LIN {X 0,Y 216.789,Z 515.517,A -85,B 0,C 180,E1 -25716.63,E2 -25716.63} C_VEL
LIN {X 0,Y 214.368,Z 508.219,A -85,B 0,C 180,E1 -25719.47,E2 -25719.47} C_VEL
LIN {X 0,Y 212.087,Z 502.265,A -85,B 0,C 180,E1 -25722.649,E2 -25722.649} C_VEL
LIN {X 0,Y 210.813,Z 499.684,A -85,B 0,C 180,E1 -25724.747,E2 -25724.747} C_VEL
LIN {X 0,Y 209.329,Z 496.442,A -85,B 0,C 180,E1 -25728.011,E2 -25728.011} C_VEL
LIN {X 0,Y 208.054,Z 493.301,A -85,B 0,C 180,E1 -25734.185,E2 -25734.185} C_VEL
LIN {X 0,Y 208.091,Z 492.674,A -85,B 0,C 180,E1 -25735.157,E2 -25735.157} C_VEL
LIN {X 0,Y 208.128,Z 492.743,A -85,B 0,C 180,E1 -25736.371,E2 -25736.371} C_VEL
LIN {X 0,Y 208.764,Z 495.592,A -85,B 0,C 180,E1 -25740.845,E2 -25740.845} C_VEL
LIN {X 0,Y 209.557,Z 496.767,A -85,B 0,C 180,E1 -25743.005,E2 -25743.005} C_VEL
LIN {X 0,Y 211.535,Z 500.908,A -85,B 0,C 180,E1 -25746.918,E2 -25746.918} C_VEL
LIN {X 0,Y 213.432,Z 504.886,A -85,B 0,C 180,E1 -25749.672,E2 -25749.672} C_VEL
LIN {X 0,Y 216.61,Z 511.711,A -85,B 0,C 180,E1 -25753.307,E2 -25753.307} C_VEL
LIN {X 0,Y 216.993,Z 512.62,A -85,B 0,C 180,E1 -25753.702,E2 -25753.702} C_VEL
LIN {X 0,Y 213.346,Z 546.935,A -85,B 0,C 180,E1 -25754.491,E2 -25754.491} C_VEL
LIN {X 0,Y 210.473,Z 562.769,A -85,B 0,C 180,E1 -25755.095,E2 -25755.095} C_VEL
LIN {X 0,Y 206.526,Z 577.358,A -85,B 0,C 180,E1 -25755.798,E2 -25755.798} C_VEL
LIN {X 0,Y 201.851,Z 590.9,A -85,B 0,C 180,E1 -25756.766,E2 -25756.766} C_VEL
LIN {X 0,Y 195.793,Z 604.759,A -85,B 0,C 180,E1 -25757.969,E2 -25757.969} C_VEL
LIN {X 0,Y 188.994,Z 617.85,A -85,B 0,C 180,E1 -25759.554,E2 -25759.554} C_VEL
LIN {X 0,Y 181.962,Z 629.225,A -85,B 0,C 180,E1 -25761.284,E2 -25761.284} C_VEL
LIN {X 0,Y 174.302,Z 639.946,A -85,B 0,C 180,E1 -25763.358,E2 -25763.358} C_VEL
LIN {X 0,Y 166.007,Z 650.074,A -85,B 0,C 180,E1 -25765.89,E2 -25765.89} C_VEL
LIN {X 0,Y 158.032,Z 658.675,A -85,B 0,C 180,E1 -25768.692,E2 -25768.692} C_VEL
LIN {X 0,Y 149.549,Z 666.826,A -85,B 0,C 180,E1 -25772.231,E2 -25772.231} C_VEL
LIN {X 0,Y 140.342,Z 674.616,A -85,B 0,C 180,E1 -25776.938,E2 -25776.938} C_VEL
LIN {X 0,Y 132.458,Z 680.534,A -85,B 0,C 180,E1 -25782.028,E2 -25782.028} C_VEL
LIN {X 0,Y 125.577,Z 685.126,A -85,B 0,C 180,E1 -25787.81,E2 -25787.81} C_VEL
LIN {X 0,Y 120.021,Z 688.366,A -85,B 0,C 180,E1 -25794.157,E2 -25794.157} C_VEL
LIN {X 0,Y 115.906,Z 690.342,A -85,B 0,C 180,E1 -25800.982,E2 -25800.982} C_VEL
LIN {X 0,Y 113.241,Z 691.138,A -85,B 0,C 180,E1 -25808.586,E2 -25808.586} C_VEL
LIN {X 0,Y 112.042,Z 690.745,A -85,B 0,C 180,E1 -25815.469,E2 -25815.469} C_VEL
LIN {X 0,Y 111.999,Z 689.219,A -85,B 0,C 180,E1 -25822.791,E2 -25822.791} C_VEL
LIN {X 0,Y 112.58,Z 687.675,A -85,B 0,C 180,E1 -25827.259,E2 -25827.259} C_VEL
LIN {X 0,Y 113.611,Z 684.748,A -85,B 0,C 180,E1 -25833.547,E2 -25833.547} C_VEL
LIN {X 0,Y 115.984,Z 680.196,A -85,B 0,C 180,E1 -25840.474,E2 -25840.474} C_VEL
LIN {X 0,Y 119.742,Z 674.292,A -85,B 0,C 180,E1 -25847.066,E2 -25847.066} C_VEL
LIN {X 0,Y 124.77,Z 666.872,A -85,B 0,C 180,E1 -25853.222,E2 -25853.222} C_VEL
LIN {X 0,Y 130.986,Z 657.702,A -85,B 0,C 180,E1 -25858.875,E2 -25858.875} C_VEL
LIN {X 0,Y 137.317,Z 647.92,A -85,B 0,C 180,E1 -25863.381,E2 -25863.381} C_VEL
LIN {X 0,Y 143.335,Z 637.901,A -85,B 0,C 180,E1 -25866.916,E2 -25866.916} C_VEL
LIN {X 0,Y 149.792,Z 626.003,A -85,B 0,C 180,E1 -25870.175,E2 -25870.175} C_VEL
LIN {X 0,Y 155.513,Z 614.116,A -85,B 0,C 180,E1 -25872.679,E2 -25872.679} C_VEL
LIN {X 0,Y 160.824,Z 601.272,A -85,B 0,C 180,E1 -25874.803,E2 -25874.803} C_VEL
LIN {X 0,Y 165.697,Z 587.197,A -85,B 0,C 180,E1 -25876.582,E2 -25876.582} C_VEL
LIN {X 0,Y 169.701,Z 572.604,A -85,B 0,C 180,E1 -25877.976,E2 -25877.976} C_VEL
LIN {X 0,Y 172.855,Z 557.467,A -85,B 0,C 180,E1 -25879.001,E2 -25879.001} C_VEL
LIN {X 0,Y 174.998,Z 541.593,A -85,B 0,C 180,E1 -25879.734,E2 -25879.734} C_VEL
LIN {X 0,Y 180.049,Z 484.1,A -85,B 0,C 180,E1 -25881.46,E2 -25881.46} C_VEL
LIN {X 0,Y 175.965,Z 475.406,A -85,B 0,C 180,E1 -25884.258,E2 -25884.258} C_VEL
LIN {X 0,Y 171.404,Z 466.555,A -85,B 0,C 180,E1 -25887.788,E2 -25887.788} C_VEL
LIN {X 0,Y 167.025,Z 458.934,A -85,B 0,C 180,E1 -25891.77,E2 -25891.77} C_VEL
LIN {X 0,Y 164.311,Z 454.695,A -85,B 0,C 180,E1 -25894.675,E2 -25894.675} C_VEL
LIN {X 0,Y 162.168,Z 451.296,A -85,B 0,C 180,E1 -25897.378,E2 -25897.378} C_VEL
LIN {X 0,Y 159.832,Z 447.476,A -85,B 0,C 180,E1 -25901.022,E2 -25901.022} C_VEL
LIN {X 0,Y 157.239,Z 443.804,A -85,B 0,C 180,E1 -25906.822,E2 -25906.822} C_VEL
LIN {X 0,Y 156.873,Z 442.502,A -85,B 0,C 180,E1 -25908.368,E2 -25908.368} C_VEL
LIN {X 0,Y 155.969,Z 441.952,A -85,B 0,C 180,E1 -25914.828,E2 -25914.828} C_VEL
LIN {X 0,Y 156.825,Z 442.233,A -85,B 0,C 180,E1 -25920.962,E2 -25920.962} C_VEL
LIN {X 0,Y 157.17,Z 442.777,A -85,B 0,C 180,E1 -25922.241,E2 -25922.241} C_VEL
LIN {X 0,Y 158.75,Z 446.055,A -85,B 0,C 180,E1 -25926.553,E2 -25926.553} C_VEL
LIN {X 0,Y 159.904,Z 447.505,A -85,B 0,C 180,E1 -25928.689,E2 -25928.689} C_VEL
LIN {X 0,Y 162.896,Z 452.334,A -85,B 0,C 180,E1 -25933.17,E2 -25933.17} C_VEL
LIN {X 0,Y 165.563,Z 456.628,A -85,B 0,C 180,E1 -25936.318,E2 -25936.318} C_VEL
LIN {X 0,Y 168.544,Z 461.52,A -85,B 0,C 180,E1 -25939.295,E2 -25939.295} C_VEL
LIN {X 0,Y 172.847,Z 469.132,A -85,B 0,C 180,E1 -25942.969,E2 -25942.969} C_VEL
LIN {X 0,Y 174.775,Z 473.432,A -85,B 0,C 180,E1 -25944.498,E2 -25944.498} C_VEL
LIN {X 0,Y 178.254,Z 483.137,A -85,B 0,C 180,E1 -25947.16,E2 -25947.16} C_VEL
LIN {X 0,Y 179.8,Z 487.933,A -85,B 0,C 180,E1 -25948.289,E2 -25948.289} C_VEL
LIN {X 0,Y 174.44,Z 549.298,A -85,B 0,C 180,E1 -25950.164,E2 -25950.164} C_VEL
LIN {X 0,Y 172.197,Z 564.852,A -85,B 0,C 180,E1 -25950.892,E2 -25950.892} C_VEL
LIN {X 0,Y 169.048,Z 579.136,A -85,B 0,C 180,E1 -25951.824,E2 -25951.824} C_VEL
LIN {X 0,Y 164.671,Z 593.902,A -85,B 0,C 180,E1 -25953.114,E2 -25953.114} C_VEL
LIN {X 0,Y 159.805,Z 607.528,A -85,B 0,C 180,E1 -25954.787,E2 -25954.787} C_VEL
LIN {X 0,Y 154.599,Z 619.845,A -85,B 0,C 180,E1 -25956.752,E2 -25956.752} C_VEL
LIN {X 0,Y 148.677,Z 632.077,A -85,B 0,C 180,E1 -25959.281,E2 -25959.281} C_VEL
LIN {X 0,Y 142.549,Z 643.378,A -85,B 0,C 180,E1 -25962.308,E2 -25962.308} C_VEL
LIN {X 0,Y 136.125,Z 654.072,A -85,B 0,C 180,E1 -25966.019,E2 -25966.019} C_VEL
LIN {X 0,Y 129.927,Z 663.892,A -85,B 0,C 180,E1 -25970.536,E2 -25970.536} C_VEL
LIN {X 0,Y 124.282,Z 672.283,A -85,B 0,C 180,E1 -25975.563,E2 -25975.563} C_VEL
LIN {X 0,Y 119.118,Z 680.145,A -85,B 0,C 180,E1 -25981.835,E2 -25981.835} C_VEL
LIN {X 0,Y 115.38,Z 686.373,A -85,B 0,C 180,E1 -25988.563,E2 -25988.563} C_VEL
LIN {X 0,Y 113.13,Z 691.156,A -85,B 0,C 180,E1 -25995.611,E2 -25995.611} C_VEL
LIN {X 0,Y 112.299,Z 693.751,A -85,B 0,C 180,E1 -26000.822,E2 -26000.822} C_VEL
LIN {X 0,Y 111.839,Z 694.596,A -85,B 0,C 180,E1 -26002.781,E2 -26002.781} C_VEL
LIN {X 0,Y 110.357,Z 695.619,A -85,B 0,C 180,E1 -26005.7,E2 -26005.7} C_VEL
LIN {X 0,Y 106.025,Z 697.111,A -85,B 0,C 180,E1 -26012.749,E2 -26012.749} C_VEL
LIN {X 0,Y 105.075,Z 697.517,A -85,B 0,C 180,E1 -26017.077,E2 -26017.077} C_VEL
LIN {X 0,Y 106.25,Z 697.472,A -85,B 0,C 180,E1 -26025.342,E2 -26025.342} C_VEL
LIN {X 0,Y 109.033,Z 696.206,A -85,B 0,C 180,E1 -26032.752,E2 -26032.752} C_VEL
LIN {X 0,Y 113.321,Z 693.824,A -85,B 0,C 180,E1 -26039.745,E2 -26039.745} C_VEL
LIN {X 0,Y 119.308,Z 690.289,A -85,B 0,C 180,E1 -26046.091,E2 -26046.091} C_VEL
LIN {X 0,Y 126.508,Z 685.508,A -85,B 0,C 180,E1 -26051.809,E2 -26051.809} C_VEL
LIN {X 0,Y 134.882,Z 679.357,A -85,B 0,C 180,E1 -26056.842,E2 -26056.842} C_VEL
LIN {X 0,Y 144.149,Z 671.666,A -85,B 0,C 180,E1 -26061.268,E2 -26061.268} C_VEL
LIN {X 0,Y 153.008,Z 663.486,A -85,B 0,C 180,E1 -26064.617,E2 -26064.617} C_VEL
LIN {X 0,Y 162.322,Z 653.69,A -85,B 0,C 180,E1 -26067.596,E2 -26067.596} C_VEL
LIN {X 0,Y 170.695,Z 643.685,A -85,B 0,C 180,E1 -26069.84,E2 -26069.84} C_VEL
LIN {X 0,Y 179.17,Z 631.906,A -85,B 0,C 180,E1 -26071.921,E2 -26071.921} C_VEL
LIN {X 0,Y 186.548,Z 620.052,A -85,B 0,C 180,E1 -26073.478,E2 -26073.478} C_VEL
LIN {X 0,Y 193.259,Z 607.331,A -85,B 0,C 180,E1 -26074.769,E2 -26074.769} C_VEL
LIN {X 0,Y 199.356,Z 593.456,A -85,B 0,C 180,E1 -26075.809,E2 -26075.809} C_VEL
LIN {X 0,Y 204.396,Z 579.169,A -85,B 0,C 180,E1 -26076.582,E2 -26076.582} C_VEL
LIN {X 0,Y 208.074,Z 565.488,A -85,B 0,C 180,E1 -26077.146,E2 -26077.146} C_VEL
LIN {X 0,Y 210.918,Z 549.998,A -85,B 0,C 180,E1 -26077.622,E2 -26077.622} C_VEL
LIN {X 0,Y 214.201,Z 519.191,A -85,B 0,C 180,E1 -26078.355,E2 -26078.355} C_VEL
LIN {X 0,Y 212.313,Z 513.341,A -85,B 0,C 180,E1 -26080.838,E2 -26080.838} C_VEL
LIN {X 0,Y 210.682,Z 508.732,A -85,B 0,C 180,E1 -26083.373,E2 -26083.373} C_VEL
LIN {X 0,Y 209.529,Z 506.271,A -85,B 0,C 180,E1 -26085.431,E2 -26085.431} C_VEL
LIN {X 0,Y 208.189,Z 503.256,A -85,B 0,C 180,E1 -26088.665,E2 -26088.665} C_VEL
LIN {X 0,Y 207.191,Z 500.002,A -85,B 0,C 180,E1 -26094.891,E2 -26094.891} C_VEL
LIN {X 0,Y 207.241,Z 499.914,A -85,B 0,C 180,E1 -26096.355,E2 -26096.355} C_VEL
LIN {X 0,Y 207.883,Z 502.7,A -85,B 0,C 180,E1 -26100.848,E2 -26100.848} C_VEL
LIN {X 0,Y 208.552,Z 503.807,A -85,B 0,C 180,E1 -26102.747,E2 -26102.747} C_VEL
LIN {X 0,Y 210.268,Z 507.604,A -85,B 0,C 180,E1 -26106.358,E2 -26106.358} C_VEL
LIN {X 0,Y 211.925,Z 511.286,A -85,B 0,C 180,E1 -26108.944,E2 -26108.944} C_VEL
LIN {X 0,Y 214.366,Z 516.868,A -85,B 0,C 180,E1 -26111.995,E2 -26111.995} C_VEL
LIN {X 0,Y 210.93,Z 547.937,A -85,B 0,C 180,E1 -26112.704,E2 -26112.704} C_VEL
LIN {X 0,Y 208.048,Z 563.218,A -85,B 0,C 180,E1 -26113.27,E2 -26113.27} C_VEL
LIN {X 0,Y 203.997,Z 577.848,A -85,B 0,C 180,E1 -26113.956,E2 -26113.956} C_VEL
LIN {X 0,Y 199.094,Z 591.641,A -85,B 0,C 180,E1 -26114.909,E2 -26114.909} C_VEL
LIN {X 0,Y 192.901,Z 605.395,A -85,B 0,C 180,E1 -26116.07,E2 -26116.07} C_VEL
LIN {X 0,Y 185.946,Z 618.371,A -85,B 0,C 180,E1 -26117.601,E2 -26117.601} C_VEL
LIN {X 0,Y 178.695,Z 629.723,A -85,B 0,C 180,E1 -26119.281,E2 -26119.281} C_VEL
LIN {X 0,Y 170.492,Z 640.806,A -85,B 0,C 180,E1 -26121.393,E2 -26121.393} C_VEL
LIN {X 0,Y 161.547,Z 651.244,A -85,B 0,C 180,E1 -26123.993,E2 -26123.993} C_VEL
LIN {X 0,Y 152.151,Z 660.809,A -85,B 0,C 180,E1 -26127.23,E2 -26127.23} C_VEL
LIN {X 0,Y 143.274,Z 668.711,A -85,B 0,C 180,E1 -26130.86,E2 -26130.86} C_VEL
LIN {X 0,Y 135.286,Z 675.069,A -85,B 0,C 180,E1 -26134.853,E2 -26134.853} C_VEL
LIN {X 0,Y 127.621,Z 680.518,A -85,B 0,C 180,E1 -26139.559,E2 -26139.559} C_VEL
LIN {X 0,Y 120.208,Z 685.162,A -85,B 0,C 180,E1 -26145.446,E2 -26145.446} C_VEL
LIN {X 0,Y 114.115,Z 688.45,A -85,B 0,C 180,E1 -26151.985,E2 -26151.985} C_VEL
LIN {X 0,Y 109.539,Z 690.489,A -85,B 0,C 180,E1 -26159.118,E2 -26159.118} C_VEL
LIN {X 0,Y 106.295,Z 691.369,A -85,B 0,C 180,E1 -26167.772,E2 -26167.772} C_VEL
LIN {X 0,Y 105.042,Z 691.015,A -85,B 0,C 180,E1 -26174.477,E2 -26174.477} C_VEL
LIN {X 0,Y 104.859,Z 689.549,A -85,B 0,C 180,E1 -26182.297,E2 -26182.297} C_VEL
LIN {X 0,Y 105.519,Z 687.844,A -85,B 0,C 180,E1 -26187.568,E2 -26187.568} C_VEL
LIN {X 0,Y 107.003,Z 684.119,A -85,B 0,C 180,E1 -26195.654,E2 -26195.654} C_VEL
LIN {X 0,Y 109.917,Z 679.324,A -85,B 0,C 180,E1 -26202.932,E2 -26202.932} C_VEL
LIN {X 0,Y 114.167,Z 673.145,A -85,B 0,C 180,E1 -26209.79,E2 -26209.79} C_VEL
LIN {X 0,Y 119.837,Z 665.382,A -85,B 0,C 180,E1 -26216.094,E2 -26216.094} C_VEL
LIN {X 0,Y 125.75,Z 657.124,A -85,B 0,C 180,E1 -26221.13,E2 -26221.13} C_VEL
LIN {X 0,Y 132.488,Z 647.183,A -85,B 0,C 180,E1 -26225.698,E2 -26225.698} C_VEL
LIN {X 0,Y 138.858,Z 637.022,A -85,B 0,C 180,E1 -26229.247,E2 -26229.247} C_VEL
LIN {X 0,Y 145.635,Z 624.903,A -85,B 0,C 180,E1 -26232.502,E2 -26232.502} C_VEL
LIN {X 0,Y 152.228,Z 611.414,A -85,B 0,C 180,E1 -26235.221,E2 -26235.221} C_VEL
LIN {X 0,Y 157.794,Z 597.924,A -85,B 0,C 180,E1 -26237.299,E2 -26237.299} C_VEL
LIN {X 0,Y 162.516,Z 583.963,A -85,B 0,C 180,E1 -26238.946,E2 -26238.946} C_VEL
LIN {X 0,Y 166.4,Z 569.598,A -85,B 0,C 180,E1 -26240.189,E2 -26240.189} C_VEL
LIN {X 0,Y 169.465,Z 554.058,A -85,B 0,C 180,E1 -26241.159,E2 -26241.159} C_VEL
LIN {X 0,Y 171.416,Z 538.62,A -85,B 0,C 180,E1 -26241.773,E2 -26241.773} C_VEL
LIN {X 0,Y 175.994,Z 487.072,A -85,B 0,C 180,E1 -26243.323,E2 -26243.323} C_VEL
LIN {X 0,Y 172.455,Z 479.342,A -85,B 0,C 180,E1 -26245.982,E2 -26245.982} C_VEL
LIN {X 0,Y 168.495,Z 471.452,A -85,B 0,C 180,E1 -26249.338,E2 -26249.338} C_VEL
LIN {X 0,Y 164.672,Z 464.588,A -85,B 0,C 180,E1 -26253.133,E2 -26253.133} C_VEL
LIN {X 0,Y 162.514,Z 461.004,A -85,B 0,C 180,E1 -26255.64,E2 -26255.64} C_VEL
LIN {X 0,Y 160.524,Z 457.695,A -85,B 0,C 180,E1 -26258.347,E2 -26258.347} C_VEL
LIN {X 0,Y 158.412,Z 454.115,A -85,B 0,C 180,E1 -26261.906,E2 -26261.906} C_VEL
LIN {X 0,Y 156.152,Z 450.578,A -85,B 0,C 180,E1 -26267.489,E2 -26267.489} C_VEL
LIN {X 0,Y 155.842,Z 449.447,A -85,B 0,C 180,E1 -26268.949,E2 -26268.949} C_VEL
LIN {X 0,Y 155.264,Z 448.928,A -85,B 0,C 180,E1 -26277.404,E2 -26277.404} C_VEL
LIN {X 0,Y 156.04,Z 449.33,A -85,B 0,C 180,E1 -26281.289,E2 -26281.289} C_VEL
LIN {X 0,Y 157.476,Z 452.718,A -85,B 0,C 180,E1 -26285.762,E2 -26285.762} C_VEL
LIN {X 0,Y 158.654,Z 454.353,A -85,B 0,C 180,E1 -26288.116,E2 -26288.116} C_VEL
LIN {X 0,Y 161.389,Z 459.036,A -85,B 0,C 180,E1 -26292.469,E2 -26292.469} C_VEL
LIN {X 0,Y 163.92,Z 463.28,A -85,B 0,C 180,E1 -26295.622,E2 -26295.622} C_VEL
LIN {X 0,Y 167.147,Z 468.9,A -85,B 0,C 180,E1 -26298.99,E2 -26298.99} C_VEL
LIN {X 0,Y 171,Z 476.238,A -85,B 0,C 180,E1 -26302.423,E2 -26302.423} C_VEL
LIN {X 0,Y 174.282,Z 485.477,A -85,B 0,C 180,E1 -26305.199,E2 -26305.199} C_VEL
LIN {X 0,Y 175.775,Z 490.371,A -85,B 0,C 180,E1 -26306.41,E2 -26306.41} C_VEL
LIN {X 0,Y 171.342,Z 540.726,A -85,B 0,C 180,E1 -26307.941,E2 -26307.941} C_VEL
LIN {X 0,Y 169.414,Z 557.45,A -85,B 0,C 180,E1 -26308.561,E2 -26308.561} C_VEL
LIN {X 0,Y 166.412,Z 572.985,A -85,B 0,C 180,E1 -26309.419,E2 -26309.419} C_VEL
LIN {X 0,Y 162.582,Z 587.033,A -85,B 0,C 180,E1 -26310.475,E2 -26310.475} C_VEL
LIN {X 0,Y 158.178,Z 600.069,A -85,B 0,C 180,E1 -26311.816,E2 -26311.816} C_VEL
LIN {X 0,Y 152.961,Z 613.236,A -85,B 0,C 180,E1 -26313.662,E2 -26313.662} C_VEL
LIN {X 0,Y 147.305,Z 625.255,A -85,B 0,C 180,E1 -26315.798,E2 -26315.798} C_VEL
LIN {X 0,Y 140.693,Z 637.61,A -85,B 0,C 180,E1 -26318.692,E2 -26318.692} C_VEL
LIN {X 0,Y 134.437,Z 648.011,A -85,B 0,C 180,E1 -26321.845,E2 -26321.845} C_VEL
LIN {X 0,Y 128.173,Z 657.582,A -85,B 0,C 180,E1 -26325.63,E2 -26325.63} C_VEL
LIN {X 0,Y 121.791,Z 667.045,A -85,B 0,C 180,E1 -26330.597,E2 -26330.597} C_VEL
LIN {X 0,Y 116.134,Z 674.858,A -85,B 0,C 180,E1 -26335.959,E2 -26335.959} C_VEL
LIN {X 0,Y 111.718,Z 681.228,A -85,B 0,C 180,E1 -26341.726,E2 -26341.726} C_VEL
LIN {X 0,Y 107.962,Z 687.25,A -85,B 0,C 180,E1 -26349.02,E2 -26349.02} C_VEL
LIN {X 0,Y 106.204,Z 690.764,A -85,B 0,C 180,E1 -26354.651,E2 -26354.651} C_VEL
LIN {X 0,Y 105.126,Z 694.276,A -85,B 0,C 180,E1 -26362.316,E2 -26362.316} C_VEL
LIN {X 0,Y 105.08,Z 695.56,A -85,B 0,C 180,E1 -26366.165,E2 -26366.165} C_VEL
LIN {X 0,Y 105.229,Z 696.538,A -85,B 0,C 180,E1 -26370,E2 -26370} C_VEL
LIN {X 0,Y 105.075,Z 697.517,A -85,B 0,C 180,E1 -26377.077,E2 -26377.077} C_VEL
LIN {X 0,Y 104.69,Z 697.712,A -85,B 0,C 180,E1 -26380.291,E2 -26380.291} C_VEL
LIN {X 0,Y 102.814,Z 697.532,A -85,B 0,C 180,E1 -26385.668,E2 -26385.668} C_VEL
LIN {X 0,Y 101.74,Z 696.955,A -85,B 0,C 180,E1 -26390.087,E2 -26390.087} C_VEL
LIN {X 0,Y 102.088,Z 696.277,A -85,B 0,C 180,E1 -26393.399,E2 -26393.399} C_VEL
LIN {X 0,Y 102.536,Z 696.006,A -85,B 0,C 180,E1 -26394.468,E2 -26394.468} C_VEL
LIN {X 0,Y 107.178,Z 693.724,A -85,B 0,C 180,E1 -26401.64,E2 -26401.64} C_VEL
LIN {X 0,Y 113.605,Z 690.245,A -85,B 0,C 180,E1 -26408.216,E2 -26408.216} C_VEL
LIN {X 0,Y 121.286,Z 685.524,A -85,B 0,C 180,E1 -26414.055,E2 -26414.055} C_VEL
LIN {X 0,Y 130.098,Z 679.424,A -85,B 0,C 180,E1 -26419.138,E2 -26419.138} C_VEL
LIN {X 0,Y 139.809,Z 671.801,A -85,B 0,C 180,E1 -26423.542,E2 -26423.542} C_VEL
LIN {X 0,Y 149,Z 663.673,A -85,B 0,C 180,E1 -26426.848,E2 -26426.848} C_VEL
LIN {X 0,Y 158.638,Z 653.96,A -85,B 0,C 180,E1 -26429.756,E2 -26429.756} C_VEL
LIN {X 0,Y 167.252,Z 644.052,A -85,B 0,C 180,E1 -26431.937,E2 -26431.937} C_VEL
LIN {X 0,Y 176.207,Z 632.006,A -85,B 0,C 180,E1 -26434.021,E2 -26434.021} C_VEL
LIN {X 0,Y 184.274,Z 619.396,A -85,B 0,C 180,E1 -26435.584,E2 -26435.584} C_VEL
LIN {X 0,Y 191.125,Z 606.582,A -85,B 0,C 180,E1 -26436.823,E2 -26436.823} C_VEL
LIN {X 0,Y 197.359,Z 592.568,A -85,B 0,C 180,E1 -26437.799,E2 -26437.799} C_VEL
LIN {X 0,Y 202.489,Z 578.078,A -85,B 0,C 180,E1 -26438.53,E2 -26438.53} C_VEL
LIN {X 0,Y 206.431,Z 563.112,A -85,B 0,C 180,E1 -26439.098,E2 -26439.098} C_VEL
LIN {X 0,Y 209.203,Z 547.133,A -85,B 0,C 180,E1 -26439.546,E2 -26439.546} C_VEL
LIN {X 0,Y 211.818,Z 523.026,A -85,B 0,C 180,E1 -26440.093,E2 -26440.093} C_VEL
LIN {X 0,Y 210.195,Z 517.831,A -85,B 0,C 180,E1 -26442.551,E2 -26442.551} C_VEL
LIN {X 0,Y 209.151,Z 514.767,A -85,B 0,C 180,E1 -26444.407,E2 -26444.407} C_VEL
LIN {X 0,Y 208.02,Z 512.33,A -85,B 0,C 180,E1 -26446.694,E2 -26446.694} C_VEL
LIN {X 0,Y 207.182,Z 510.194,A -85,B 0,C 180,E1 -26449.017,E2 -26449.017} C_VEL
LIN {X 0,Y 206.32,Z 507.013,A -85,B 0,C 180,E1 -26455.116,E2 -26455.116} C_VEL
LIN {X 0,Y 206.351,Z 507.112,A -85,B 0,C 180,E1 -26456.339,E2 -26456.339} C_VEL
LIN {X 0,Y 207.117,Z 509.982,A -85,B 0,C 180,E1 -26461.216,E2 -26461.216} C_VEL
LIN {X 0,Y 207.59,Z 510.994,A -85,B 0,C 180,E1 -26462.608,E2 -26462.608} C_VEL
LIN {X 0,Y 209.025,Z 514.28,A -85,B 0,C 180,E1 -26465.79,E2 -26465.79} C_VEL
LIN {X 0,Y 210.584,Z 517.995,A -85,B 0,C 180,E1 -26468.397,E2 -26468.397} C_VEL
LIN {X 0,Y 211.931,Z 521.305,A -85,B 0,C 180,E1 -26470.269,E2 -26470.269} C_VEL
LIN {X 0,Y 208.804,Z 548.452,A -85,B 0,C 180,E1 -26470.867,E2 -26470.867} C_VEL
LIN {X 0,Y 205.723,Z 564.159,A -85,B 0,C 180,E1 -26471.435,E2 -26471.435} C_VEL
LIN {X 0,Y 201.706,Z 578.27,A -85,B 0,C 180,E1 -26472.068,E2 -26472.068} C_VEL
LIN {X 0,Y 196.522,Z 592.439,A -85,B 0,C 180,E1 -26473.009,E2 -26473.009} C_VEL
LIN {X 0,Y 190.228,Z 606.026,A -85,B 0,C 180,E1 -26474.114,E2 -26474.114} C_VEL
LIN {X 0,Y 183.143,Z 618.857,A -85,B 0,C 180,E1 -26475.583,E2 -26475.583} C_VEL
LIN {X 0,Y 174.908,Z 631.315,A -85,B 0,C 180,E1 -26477.388,E2 -26477.388} C_VEL
LIN {X 0,Y 165.97,Z 642.803,A -85,B 0,C 180,E1 -26479.58,E2 -26479.58} C_VEL
LIN {X 0,Y 155.859,Z 653.895,A -85,B 0,C 180,E1 -26482.424,E2 -26482.424} C_VEL
LIN {X 0,Y 146.565,Z 662.751,A -85,B 0,C 180,E1 -26485.568,E2 -26485.568} C_VEL
LIN {X 0,Y 137.116,Z 670.597,A -85,B 0,C 180,E1 -26489.384,E2 -26489.384} C_VEL
LIN {X 0,Y 127.512,Z 677.588,A -85,B 0,C 180,E1 -26494.234,E2 -26494.234} C_VEL
LIN {X 0,Y 118.895,Z 683.012,A -85,B 0,C 180,E1 -26499.786,E2 -26499.786} C_VEL
LIN {X 0,Y 111.529,Z 687.023,A -85,B 0,C 180,E1 -26506.119,E2 -26506.119} C_VEL
LIN {X 0,Y 105.669,Z 689.739,A -85,B 0,C 180,E1 -26513.231,E2 -26513.231} C_VEL
LIN {X 0,Y 101.355,Z 691.238,A -85,B 0,C 180,E1 -26520.963,E2 -26520.963} C_VEL
LIN {X 0,Y 98.808,Z 691.557,A -85,B 0,C 180,E1 -26529.168,E2 -26529.168} C_VEL
LIN {X 0,Y 97.704,Z 690.726,A -85,B 0,C 180,E1 -26537.538,E2 -26537.538} C_VEL
LIN {X 0,Y 98.108,Z 688.727,A -85,B 0,C 180,E1 -26545.892,E2 -26545.892} C_VEL
LIN {X 0,Y 98.662,Z 687.274,A -85,B 0,C 180,E1 -26550,E2 -26550} C_VEL
LIN {X 0,Y 100.537,Z 683.478,A -85,B 0,C 180,E1 -26558.037,E2 -26558.037} C_VEL
LIN {X 0,Y 104.018,Z 678.396,A -85,B 0,C 180,E1 -26565.68,E2 -26565.68} C_VEL
LIN {X 0,Y 108.925,Z 671.906,A -85,B 0,C 180,E1 -26572.776,E2 -26572.776} C_VEL
LIN {X 0,Y 115.202,Z 663.803,A -85,B 0,C 180,E1 -26579.213,E2 -26579.213} C_VEL
LIN {X 0,Y 121.701,Z 655.159,A -85,B 0,C 180,E1 -26584.267,E2 -26584.267} C_VEL
LIN {X 0,Y 128.973,Z 644.774,A -85,B 0,C 180,E1 -26588.805,E2 -26588.805} C_VEL
LIN {X 0,Y 135.763,Z 634.119,A -85,B 0,C 180,E1 -26592.297,E2 -26592.297} C_VEL
LIN {X 0,Y 142.962,Z 621.343,A -85,B 0,C 180,E1 -26595.465,E2 -26595.465} C_VEL
LIN {X 0,Y 149.242,Z 608.44,A -85,B 0,C 180,E1 -26597.876,E2 -26597.876} C_VEL
LIN {X 0,Y 154.401,Z 595.94,A -85,B 0,C 180,E1 -26599.679,E2 -26599.679} C_VEL
LIN {X 0,Y 159.304,Z 581.375,A -85,B 0,C 180,E1 -26601.29,E2 -26601.29} C_VEL
LIN {X 0,Y 163.331,Z 566.08,A -85,B 0,C 180,E1 -26602.5,E2 -26602.5} C_VEL
LIN {X 0,Y 166.173,Z 550.893,A -85,B 0,C 180,E1 -26603.346,E2 -26603.346} C_VEL
LIN {X 0,Y 168.253,Z 532.641,A -85,B 0,C 180,E1 -26603.981,E2 -26603.981} C_VEL
LIN {X 0,Y 172.136,Z 490.174,A -85,B 0,C 180,E1 -26605.253,E2 -26605.253} C_VEL
LIN {X 0,Y 168.053,Z 481.155,A -85,B 0,C 180,E1 -26608.705,E2 -26608.705} C_VEL
LIN {X 0,Y 164.609,Z 474.255,A -85,B 0,C 180,E1 -26612.074,E2 -26612.074} C_VEL
LIN {X 0,Y 161.317,Z 468.144,A -85,B 0,C 180,E1 -26615.917,E2 -26615.917} C_VEL
LIN {X 0,Y 158.955,Z 464.15,A -85,B 0,C 180,E1 -26619.284,E2 -26619.284} C_VEL
LIN {X 0,Y 157.054,Z 460.806,A -85,B 0,C 180,E1 -26622.754,E2 -26622.754} C_VEL
LIN {X 0,Y 155.043,Z 457.148,A -85,B 0,C 180,E1 -26628.395,E2 -26628.395} C_VEL
LIN {X 0,Y 154.824,Z 456.416,A -85,B 0,C 180,E1 -26629.537,E2 -26629.537} C_VEL
LIN {X 0,Y 154.639,Z 456.053,A -85,B 0,C 180,E1 -26639.026,E2 -26639.026} C_VEL
LIN {X 0,Y 155.095,Z 456.555,A -85,B 0,C 180,E1 -26641.135,E2 -26641.135} C_VEL
LIN {X 0,Y 156.731,Z 460.125,A -85,B 0,C 180,E1 -26646.112,E2 -26646.112} C_VEL
LIN {X 0,Y 157.491,Z 461.404,A -85,B 0,C 180,E1 -26647.692,E2 -26647.692} C_VEL
LIN {X 0,Y 159.754,Z 465.419,A -85,B 0,C 180,E1 -26651.525,E2 -26651.525} C_VEL
LIN {X 0,Y 162.225,Z 469.831,A -85,B 0,C 180,E1 -26654.824,E2 -26654.824} C_VEL
LIN {X 0,Y 165.055,Z 475.021,A -85,B 0,C 180,E1 -26657.98,E2 -26657.98} C_VEL
LIN {X 0,Y 168.472,Z 482.034,A -85,B 0,C 180,E1 -26661.267,E2 -26661.267} C_VEL
LIN {X 0,Y 171.375,Z 490.819,A -85,B 0,C 180,E1 -26663.938,E2 -26663.938} C_VEL
LIN {X 0,Y 172.007,Z 493.133,A -85,B 0,C 180,E1 -26664.513,E2 -26664.513} C_VEL
LIN {X 0,Y 166.376,Z 552.178,A -85,B 0,C 180,E1 -26666.284,E2 -26666.284} C_VEL
LIN {X 0,Y 163.719,Z 567.648,A -85,B 0,C 180,E1 -26667.033,E2 -26667.033} C_VEL
LIN {X 0,Y 159.808,Z 583.037,A -85,B 0,C 180,E1 -26668.078,E2 -26668.078} C_VEL
LIN {X 0,Y 155.201,Z 596.864,A -85,B 0,C 180,E1 -26669.343,E2 -26669.343} C_VEL
LIN {X 0,Y 149.688,Z 610.704,A -85,B 0,C 180,E1 -26671.138,E2 -26671.138} C_VEL
LIN {X 0,Y 143.214,Z 624.247,A -85,B 0,C 180,E1 -26673.462,E2 -26673.462} C_VEL
LIN {X 0,Y 136.279,Z 636.732,A -85,B 0,C 180,E1 -26676.313,E2 -26676.313} C_VEL
LIN {X 0,Y 128.599,Z 648.937,A -85,B 0,C 180,E1 -26680.083,E2 -26680.083} C_VEL
LIN {X 0,Y 121.707,Z 658.981,A -85,B 0,C 180,E1 -26684.27,E2 -26684.27} C_VEL
LIN {X 0,Y 115.384,Z 667.676,A -85,B 0,C 180,E1 -26689.097,E2 -26689.097} C_VEL
LIN {X 0,Y 109.48,Z 675.337,A -85,B 0,C 180,E1 -26694.707,E2 -26694.707} C_VEL
LIN {X 0,Y 104.172,Z 682.484,A -85,B 0,C 180,E1 -26701.819,E2 -26701.819} C_VEL
LIN {X 0,Y 100.526,Z 688.094,A -85,B 0,C 180,E1 -26709.539,E2 -26709.539} C_VEL
LIN {X 0,Y 98.483,Z 692.315,A -85,B 0,C 180,E1 -26717.638,E2 -26717.638} C_VEL
LIN {X 0,Y 97.99,Z 695.251,A -85,B 0,C 180,E1 -26725.887,E2 -26725.887} C_VEL
LIN {X 0,Y 98.141,Z 696.256,A -85,B 0,C 180,E1 -26730,E2 -26730} C_VEL
LIN {X 0,Y 97.988,Z 697.242,A -85,B 0,C 180,E1 -26737.192,E2 -26737.192} C_VEL
LIN {X 0,Y 98.507,Z 697.457,A -85,B 0,C 180,E1 -26742.359,E2 -26742.359} C_VEL
LIN {X 0,Y 100.662,Z 696.793,A -85,B 0,C 180,E1 -26750.431,E2 -26750.431} C_VEL
LIN {X 0,Y 102.536,Z 696.006,A -85,B 0,C 180,E1 -26754.468,E2 -26754.468} C_VEL
LIN {X 0,Y 103.673,Z 695.202,A -85,B 0,C 180,E1 -26757.655,E2 -26757.655} C_VEL
LIN {X 0,Y 104.516,Z 693.542,A -85,B 0,C 180,E1 -26763.023,E2 -26763.023} C_VEL
LIN {X 0,Y 105.685,Z 691.951,A -85,B 0,C 180,E1 -26767.217,E2 -26767.217} C_VEL
LIN {X 0,Y 107.622,Z 690.485,A -85,B 0,C 180,E1 -26770.109,E2 -26770.109} C_VEL
LIN {X 0,Y 108.554,Z 689.922,A -85,B 0,C 180,E1 -26770.981,E2 -26770.981} C_VEL
LIN {X 0,Y 116.272,Z 685.529,A -85,B 0,C 180,E1 -26776.497,E2 -26776.497} C_VEL
LIN {X 0,Y 125.539,Z 679.474,A -85,B 0,C 180,E1 -26781.606,E2 -26781.606} C_VEL
LIN {X 0,Y 135.697,Z 671.918,A -85,B 0,C 180,E1 -26785.962,E2 -26785.962} C_VEL
LIN {X 0,Y 146.621,Z 662.624,A -85,B 0,C 180,E1 -26789.632,E2 -26789.632} C_VEL
LIN {X 0,Y 156.632,Z 652.747,A -85,B 0,C 180,E1 -26792.396,E2 -26792.396} C_VEL
LIN {X 0,Y 167.012,Z 640.811,A -85,B 0,C 180,E1 -26794.788,E2 -26794.788} C_VEL
LIN {X 0,Y 176.018,Z 628.482,A -85,B 0,C 180,E1 -26796.684,E2 -26796.684} C_VEL
LIN {X 0,Y 183.818,Z 616.127,A -85,B 0,C 180,E1 -26797.997,E2 -26797.997} C_VEL
LIN {X 0,Y 190.826,Z 602.657,A -85,B 0,C 180,E1 -26799.155,E2 -26799.155} C_VEL
LIN {X 0,Y 196.816,Z 588.708,A -85,B 0,C 180,E1 -26799.981,E2 -26799.981} C_VEL
LIN {X 0,Y 201.952,Z 573.212,A -85,B 0,C 180,E1 -26800.684,E2 -26800.684} C_VEL
LIN {X 0,Y 205.699,Z 557.544,A -85,B 0,C 180,E1 -26801.164,E2 -26801.164} C_VEL
LIN {X 0,Y 208.137,Z 540.924,A -85,B 0,C 180,E1 -26801.546,E2 -26801.546} C_VEL
LIN {X 0,Y 209.602,Z 527.004,A -85,B 0,C 180,E1 -26801.885,E2 -26801.885} C_VEL
LIN {X 0,Y 208.043,Z 521.793,A -85,B 0,C 180,E1 -26804.73,E2 -26804.73} C_VEL
LIN {X 0,Y 207.139,Z 519.636,A -85,B 0,C 180,E1 -26806.637,E2 -26806.637} C_VEL
LIN {X 0,Y 206.242,Z 517.189,A -85,B 0,C 180,E1 -26809.199,E2 -26809.199} C_VEL
LIN {X 0,Y 205.44,Z 514.146,A -85,B 0,C 180,E1 -26815.095,E2 -26815.095} C_VEL
LIN {X 0,Y 205.464,Z 514.361,A -85,B 0,C 180,E1 -26816.446,E2 -26816.446} C_VEL
LIN {X 0,Y 206.237,Z 517.083,A -85,B 0,C 180,E1 -26821.221,E2 -26821.221} C_VEL
LIN {X 0,Y 207.691,Z 520.642,A -85,B 0,C 180,E1 -26824.975,E2 -26824.975} C_VEL
LIN {X 0,Y 209.19,Z 524.506,A -85,B 0,C 180,E1 -26827.724,E2 -26827.724} C_VEL
LIN {X 0,Y 209.662,Z 525.825,A -85,B 0,C 180,E1 -26828.481,E2 -26828.481} C_VEL
LIN {X 0,Y 206.798,Z 549.504,A -85,B 0,C 180,E1 -26829.003,E2 -26829.003} C_VEL
LIN {X 0,Y 203.721,Z 564.642,A -85,B 0,C 180,E1 -26829.527,E2 -26829.527} C_VEL
LIN {X 0,Y 199.579,Z 578.844,A -85,B 0,C 180,E1 -26830.142,E2 -26830.142} C_VEL
LIN {X 0,Y 194.132,Z 593.297,A -85,B 0,C 180,E1 -26831.069,E2 -26831.069} C_VEL
LIN {X 0,Y 187.781,Z 606.64,A -85,B 0,C 180,E1 -26832.104,E2 -26832.104} C_VEL
LIN {X 0,Y 180.522,Z 619.42,A -85,B 0,C 180,E1 -26833.51,E2 -26833.51} C_VEL
LIN {X 0,Y 172.087,Z 631.81,A -85,B 0,C 180,E1 -26835.239,E2 -26835.239} C_VEL
LIN {X 0,Y 163.657,Z 642.346,A -85,B 0,C 180,E1 -26837.158,E2 -26837.158} C_VEL
LIN {X 0,Y 154.686,Z 652.071,A -85,B 0,C 180,E1 -26839.481,E2 -26839.481} C_VEL
LIN {X 0,Y 144.585,Z 661.568,A -85,B 0,C 180,E1 -26842.549,E2 -26842.549} C_VEL
LIN {X 0,Y 134.974,Z 669.413,A -85,B 0,C 180,E1 -26846.078,E2 -26846.078} C_VEL
LIN {X 0,Y 125.805,Z 675.959,A -85,B 0,C 180,E1 -26850.186,E2 -26850.186} C_VEL
LIN {X 0,Y 116.497,Z 681.748,A -85,B 0,C 180,E1 -26855.47,E2 -26855.47} C_VEL
LIN {X 0,Y 110.159,Z 685.207,A -85,B 0,C 180,E1 -26860.041,E2 -26860.041} C_VEL
LIN {X 0,Y 102.876,Z 688.625,A -85,B 0,C 180,E1 -26866.91,E2 -26866.91} C_VEL
LIN {X 0,Y 97.205,Z 690.788,A -85,B 0,C 180,E1 -26874.662,E2 -26874.662} C_VEL
LIN {X 0,Y 93.266,Z 691.754,A -85,B 0,C 180,E1 -26883.12,E2 -26883.12} C_VEL
LIN {X 0,Y 91.138,Z 691.553,A -85,B 0,C 180,E1 -26892.034,E2 -26892.034} C_VEL
LIN {X 0,Y 90.586,Z 690.193,A -85,B 0,C 180,E1 -26901.074,E2 -26901.074} C_VEL
LIN {X 0,Y 91.396,Z 688.104,A -85,B 0,C 180,E1 -26908.562,E2 -26908.562} C_VEL
LIN {X 0,Y 92.918,Z 684.955,A -85,B 0,C 180,E1 -26916.515,E2 -26916.515} C_VEL
LIN {X 0,Y 96.129,Z 680.295,A -85,B 0,C 180,E1 -26924.826,E2 -26924.826} C_VEL
LIN {X 0,Y 100.98,Z 674.247,A -85,B 0,C 180,E1 -26932.507,E2 -26932.507} C_VEL
LIN {X 0,Y 107.306,Z 666.646,A -85,B 0,C 180,E1 -26939.42,E2 -26939.42} C_VEL
LIN {X 0,Y 113.869,Z 658.515,A -85,B 0,C 180,E1 -26944.814,E2 -26944.814} C_VEL
LIN {X 0,Y 121.3,Z 648.761,A -85,B 0,C 180,E1 -26949.593,E2 -26949.593} C_VEL
LIN {X 0,Y 128.251,Z 638.773,A -85,B 0,C 180,E1 -26953.235,E2 -26953.235} C_VEL
LIN {X 0,Y 135.586,Z 626.916,A -85,B 0,C 180,E1 -26956.526,E2 -26956.526} C_VEL
LIN {X 0,Y 142.006,Z 615.08,A -85,B 0,C 180,E1 -26959.003,E2 -26959.003} C_VEL
LIN {X 0,Y 147.948,Z 602.296,A -85,B 0,C 180,E1 -26961.066,E2 -26961.066} C_VEL
LIN {X 0,Y 153.335,Z 588.316,A -85,B 0,C 180,E1 -26962.785,E2 -26962.785} C_VEL
LIN {X 0,Y 157.764,Z 573.859,A -85,B 0,C 180,E1 -26964.117,E2 -26964.117} C_VEL
LIN {X 0,Y 161.388,Z 558.067,A -85,B 0,C 180,E1 -26965.145,E2 -26965.145} C_VEL
LIN {X 0,Y 163.641,Z 543.253,A -85,B 0,C 180,E1 -26965.8,E2 -26965.8} C_VEL
LIN {X 0,Y 168.454,Z 493.301,A -85,B 0,C 180,E1 -26967.285,E2 -26967.285} C_VEL
LIN {X 0,Y 164.508,Z 484.364,A -85,B 0,C 180,E1 -26971.04,E2 -26971.04} C_VEL
LIN {X 0,Y 161.091,Z 477.351,A -85,B 0,C 180,E1 -26974.917,E2 -26974.917} C_VEL
LIN {X 0,Y 158.862,Z 473.239,A -85,B 0,C 180,E1 -26977.935,E2 -26977.935} C_VEL
LIN {X 0,Y 157.601,Z 470.867,A -85,B 0,C 180,E1 -26979.95,E2 -26979.95} C_VEL
LIN {X 0,Y 155.851,Z 467.624,A -85,B 0,C 180,E1 -26983.361,E2 -26983.361} C_VEL
LIN {X 0,Y 153.995,Z 463.881,A -85,B 0,C 180,E1 -26989.148,E2 -26989.148} C_VEL
LIN {X 0,Y 153.811,Z 463.366,A -85,B 0,C 180,E1 -26990.201,E2 -26990.201} C_VEL
LIN {X 0,Y 153.518,Z 463.022,A -85,B 0,C 180,E1 -26997.375,E2 -26997.375} C_VEL
LIN {X 0,Y 154.077,Z 463.423,A -85,B 0,C 180,E1 -27000.551,E2 -27000.551} C_VEL
LIN {X 0,Y 155.698,Z 467.117,A -85,B 0,C 180,E1 -27005.828,E2 -27005.828} C_VEL
LIN {X 0,Y 158.258,Z 471.997,A -85,B 0,C 180,E1 -27010.716,E2 -27010.716} C_VEL
LIN {X 0,Y 160.58,Z 476.391,A -85,B 0,C 180,E1 -27014.029,E2 -27014.029} C_VEL
LIN {X 0,Y 163.378,Z 481.921,A -85,B 0,C 180,E1 -27017.347,E2 -27017.347} C_VEL
LIN {X 0,Y 165.981,Z 487.711,A -85,B 0,C 180,E1 -27020.041,E2 -27020.041} C_VEL
LIN {X 0,Y 168.318,Z 495.35,A -85,B 0,C 180,E1 -27022.407,E2 -27022.407} C_VEL
LIN {X 0,Y 168.171,Z 498.155,A -85,B 0,C 180,E1 -27022.567,E2 -27022.567} C_VEL
LIN {X 0,Y 162.778,Z 552.374,A -85,B 0,C 180,E1 -27024.163,E2 -27024.163} C_VEL
LIN {X 0,Y 160.04,Z 567.707,A -85,B 0,C 180,E1 -27024.892,E2 -27024.892} C_VEL
LIN {X 0,Y 156.212,Z 582.458,A -85,B 0,C 180,E1 -27025.867,E2 -27025.867} C_VEL
LIN {X 0,Y 151.103,Z 597.268,A -85,B 0,C 180,E1 -27027.185,E2 -27027.185} C_VEL
LIN {X 0,Y 145.747,Z 610.227,A -85,B 0,C 180,E1 -27028.828,E2 -27028.828} C_VEL
LIN {X 0,Y 139.357,Z 623.173,A -85,B 0,C 180,E1 -27030.981,E2 -27030.981} C_VEL
LIN {X 0,Y 132.804,Z 634.731,A -85,B 0,C 180,E1 -27033.541,E2 -27033.541} C_VEL
LIN {X 0,Y 125.311,Z 646.388,A -85,B 0,C 180,E1 -27036.945,E2 -27036.945} C_VEL
LIN {X 0,Y 117.923,Z 656.652,A -85,B 0,C 180,E1 -27040.962,E2 -27040.962} C_VEL
LIN {X 0,Y 111.018,Z 665.787,A -85,B 0,C 180,E1 -27045.864,E2 -27045.864} C_VEL
LIN {X 0,Y 104.522,Z 673.752,A -85,B 0,C 180,E1 -27051.54,E2 -27051.54} C_VEL
LIN {X 0,Y 98.589,Z 681.124,A -85,B 0,C 180,E1 -27058.804,E2 -27058.804} C_VEL
LIN {X 0,Y 94.68,Z 686.402,A -85,B 0,C 180,E1 -27065.904,E2 -27065.904} C_VEL
LIN {X 0,Y 92.434,Z 689.974,A -85,B 0,C 180,E1 -27072.294,E2 -27072.294} C_VEL
LIN {X 0,Y 90.995,Z 693.601,A -85,B 0,C 180,E1 -27081.114,E2 -27081.114} C_VEL
LIN {X 0,Y 90.895,Z 694.941,A -85,B 0,C 180,E1 -27085.565,E2 -27085.565} C_VEL
LIN {X 0,Y 91.044,Z 695.973,A -85,B 0,C 180,E1 -27090,E2 -27090} C_VEL
LIN {X 0,Y 91.018,Z 697.109,A -85,B 0,C 180,E1 -27098.884,E2 -27098.884} C_VEL
LIN {X 0,Y 92.522,Z 697.057,A -85,B 0,C 180,E1 -27107.688,E2 -27107.688} C_VEL
LIN {X 0,Y 95.958,Z 695.895,A -85,B 0,C 180,E1 -27116.068,E2 -27116.068} C_VEL
LIN {X 0,Y 101.159,Z 693.623,A -85,B 0,C 180,E1 -27123.766,E2 -27123.766} C_VEL
LIN {X 0,Y 108.554,Z 689.922,A -85,B 0,C 180,E1 -27130.981,E2 -27130.981} C_VEL
LIN {X 0,Y 111.153,Z 688.246,A -85,B 0,C 180,E1 -27133.601,E2 -27133.601} C_VEL
LIN {X 0,Y 114.437,Z 685.213,A -85,B 0,C 180,E1 -27138.108,E2 -27138.108} C_VEL
LIN {X 0,Y 117.327,Z 682.522,A -85,B 0,C 180,E1 -27141.522,E2 -27141.522} C_VEL
LIN {X 0,Y 120.262,Z 680.203,A -85,B 0,C 180,E1 -27143.738,E2 -27143.738} C_VEL
LIN {X 0,Y 121.447,Z 679.363,A -85,B 0,C 180,E1 -27144.372,E2 -27144.372} C_VEL
LIN {X 0,Y 131.838,Z 672.031,A -85,B 0,C 180,E1 -27148.531,E2 -27148.531} C_VEL
LIN {X 0,Y 143.167,Z 662.818,A -85,B 0,C 180,E1 -27152.081,E2 -27152.081} C_VEL
LIN {X 0,Y 153.478,Z 653.021,A -85,B 0,C 180,E1 -27154.74,E2 -27154.74} C_VEL
LIN {X 0,Y 162.598,Z 643.014,A -85,B 0,C 180,E1 -27156.707,E2 -27156.707} C_VEL
LIN {X 0,Y 171.738,Z 631.245,A -85,B 0,C 180,E1 -27158.542,E2 -27158.542} C_VEL
LIN {X 0,Y 179.691,Z 619.372,A -85,B 0,C 180,E1 -27159.831,E2 -27159.831} C_VEL
LIN {X 0,Y 186.831,Z 606.649,A -85,B 0,C 180,E1 -27160.931,E2 -27160.931} C_VEL
LIN {X 0,Y 193.288,Z 592.767,A -85,B 0,C 180,E1 -27161.789,E2 -27161.789} C_VEL
LIN {X 0,Y 198.584,Z 578.484,A -85,B 0,C 180,E1 -27162.428,E2 -27162.428} C_VEL
LIN {X 0,Y 202.534,Z 564.431,A -85,B 0,C 180,E1 -27162.908,E2 -27162.908} C_VEL
LIN {X 0,Y 205.448,Z 549.382,A -85,B 0,C 180,E1 -27163.302,E2 -27163.302} C_VEL
LIN {X 0,Y 207.591,Z 531.323,A -85,B 0,C 180,E1 -27163.682,E2 -27163.682} C_VEL
LIN {X 0,Y 206.633,Z 527.918,A -85,B 0,C 180,E1 -27165.725,E2 -27165.725} C_VEL
LIN {X 0,Y 205.219,Z 524.095,A -85,B 0,C 180,E1 -27169.643,E2 -27169.643} C_VEL
LIN {X 0,Y 204.557,Z 521.295,A -85,B 0,C 180,E1 -27175.11,E2 -27175.11} C_VEL
LIN {X 0,Y 204.577,Z 521.531,A -85,B 0,C 180,E1 -27176.431,E2 -27176.431} C_VEL
LIN {X 0,Y 205.46,Z 524.522,A -85,B 0,C 180,E1 -27181.593,E2 -27181.593} C_VEL
LIN {X 0,Y 206.769,Z 528.107,A -85,B 0,C 180,E1 -27184.998,E2 -27184.998} C_VEL
LIN {X 0,Y 207.624,Z 530.468,A -85,B 0,C 180,E1 -27186.682,E2 -27186.682} C_VEL
LIN {X 0,Y 205.094,Z 550.207,A -85,B 0,C 180,E1 -27187.095,E2 -27187.095} C_VEL
LIN {X 0,Y 201.807,Z 565.756,A -85,B 0,C 180,E1 -27187.625,E2 -27187.625} C_VEL
LIN {X 0,Y 197.722,Z 579.339,A -85,B 0,C 180,E1 -27188.175,E2 -27188.175} C_VEL
LIN {X 0,Y 192.149,Z 593.753,A -85,B 0,C 180,E1 -27189.051,E2 -27189.051} C_VEL
LIN {X 0,Y 185.572,Z 607.238,A -85,B 0,C 180,E1 -27190.043,E2 -27190.043} C_VEL
LIN {X 0,Y 178.171,Z 619.933,A -85,B 0,C 180,E1 -27191.376,E2 -27191.376} C_VEL
LIN {X 0,Y 169.52,Z 632.299,A -85,B 0,C 180,E1 -27193.026,E2 -27193.026} C_VEL
LIN {X 0,Y 160.097,Z 643.695,A -85,B 0,C 180,E1 -27195.036,E2 -27195.036} C_VEL
LIN {X 0,Y 150.875,Z 653.24,A -85,B 0,C 180,E1 -27197.269,E2 -27197.269} C_VEL
LIN {X 0,Y 141.915,Z 661.32,A -85,B 0,C 180,E1 -27199.791,E2 -27199.791} C_VEL
LIN {X 0,Y 131.904,Z 669.253,A -85,B 0,C 180,E1 -27203.205,E2 -27203.205} C_VEL
LIN {X 0,Y 121.423,Z 676.399,A -85,B 0,C 180,E1 -27207.585,E2 -27207.585} C_VEL
LIN {X 0,Y 112.387,Z 681.737,A -85,B 0,C 180,E1 -27212.413,E2 -27212.413} C_VEL
LIN {X 0,Y 105.564,Z 685.23,A -85,B 0,C 180,E1 -27216.974,E2 -27216.974} C_VEL
LIN {X 0,Y 97.614,Z 688.713,A -85,B 0,C 180,E1 -27223.947,E2 -27223.947} C_VEL
LIN {X 0,Y 91.296,Z 690.938,A -85,B 0,C 180,E1 -27231.987,E2 -27231.987} C_VEL
LIN {X 0,Y 86.792,Z 691.965,A -85,B 0,C 180,E1 -27240.932,E2 -27240.932} C_VEL
LIN {X 0,Y 84.256,Z 691.822,A -85,B 0,C 180,E1 -27250.51,E2 -27250.51} C_VEL
LIN {X 0,Y 83.477,Z 690.491,A -85,B 0,C 180,E1 -27260.307,E2 -27260.307} C_VEL
LIN {X 0,Y 84.428,Z 687.983,A -85,B 0,C 180,E1 -27270,E2 -27270} C_VEL
LIN {X 0,Y 86.54,Z 684.308,A -85,B 0,C 180,E1 -27279.348,E2 -27279.348} C_VEL
LIN {X 0,Y 90.438,Z 679.36,A -85,B 0,C 180,E1 -27288.11,E2 -27288.11} C_VEL
LIN {X 0,Y 96.057,Z 673.007,A -85,B 0,C 180,E1 -27296.04,E2 -27296.04} C_VEL
LIN {X 0,Y 103.097,Z 665.062,A -85,B 0,C 180,E1 -27303.049,E2 -27303.049} C_VEL
LIN {X 0,Y 110.305,Z 656.593,A -85,B 0,C 180,E1 -27308.405,E2 -27308.405} C_VEL
LIN {X 0,Y 118.305,Z 646.408,A -85,B 0,C 180,E1 -27313.092,E2 -27313.092} C_VEL
LIN {X 0,Y 125.698,Z 635.989,A -85,B 0,C 180,E1 -27316.624,E2 -27316.624} C_VEL
LIN {X 0,Y 132.799,Z 624.668,A -85,B 0,C 180,E1 -27319.531,E2 -27319.531} C_VEL
LIN {X 0,Y 139.534,Z 612.373,A -85,B 0,C 180,E1 -27321.906,E2 -27321.906} C_VEL
LIN {X 0,Y 145.689,Z 598.959,A -85,B 0,C 180,E1 -27323.903,E2 -27323.903} C_VEL
LIN {X 0,Y 150.929,Z 585.072,A -85,B 0,C 180,E1 -27325.449,E2 -27325.449} C_VEL
LIN {X 0,Y 155.178,Z 570.831,A -85,B 0,C 180,E1 -27326.62,E2 -27326.62} C_VEL
LIN {X 0,Y 158.552,Z 555.519,A -85,B 0,C 180,E1 -27327.525,E2 -27327.525} C_VEL
LIN {X 0,Y 160.658,Z 540.75,A -85,B 0,C 180,E1 -27328.105,E2 -27328.105} C_VEL
LIN {X 0,Y 165.039,Z 496.794,A -85,B 0,C 180,E1 -27329.334,E2 -27329.334} C_VEL
LIN {X 0,Y 161.816,Z 489.085,A -85,B 0,C 180,E1 -27332.778,E2 -27332.778} C_VEL
LIN {X 0,Y 158.845,Z 482.763,A -85,B 0,C 180,E1 -27336.533,E2 -27336.533} C_VEL
LIN {X 0,Y 156.544,Z 478.048,A -85,B 0,C 180,E1 -27340.145,E2 -27340.145} C_VEL
LIN {X 0,Y 154.582,Z 474.351,A -85,B 0,C 180,E1 -27344.169,E2 -27344.169} C_VEL
LIN {X 0,Y 152.946,Z 470.432,A -85,B 0,C 180,E1 -27350.145,E2 -27350.145} C_VEL
LIN {X 0,Y 152.832,Z 470.127,A -85,B 0,C 180,E1 -27358.681,E2 -27358.681} C_VEL
LIN {X 0,Y 153.131,Z 470.584,A -85,B 0,C 180,E1 -27360.334,E2 -27360.334} C_VEL
LIN {X 0,Y 154.941,Z 474.795,A -85,B 0,C 180,E1 -27366.221,E2 -27366.221} C_VEL
LIN {X 0,Y 157.039,Z 479.093,A -85,B 0,C 180,E1 -27370.311,E2 -27370.311} C_VEL
LIN {X 0,Y 159.104,Z 483.21,A -85,B 0,C 180,E1 -27373.408,E2 -27373.408} C_VEL
LIN {X 0,Y 161.939,Z 489.293,A -85,B 0,C 180,E1 -27376.951,E2 -27376.951} C_VEL
LIN {X 0,Y 163.715,Z 493.75,A -85,B 0,C 180,E1 -27378.932,E2 -27378.932} C_VEL
LIN {X 0,Y 164.93,Z 498.179,A -85,B 0,C 180,E1 -27380.32,E2 -27380.32} C_VEL
LIN {X 0,Y 161.379,Z 535.237,A -85,B 0,C 180,E1 -27381.435,E2 -27381.435} C_VEL
LIN {X 0,Y 159.186,Z 553.98,A -85,B 0,C 180,E1 -27382.005,E2 -27382.005} C_VEL
LIN {X 0,Y 156.189,Z 569.282,A -85,B 0,C 180,E1 -27382.715,E2 -27382.715} C_VEL
LIN {X 0,Y 152.087,Z 584.151,A -85,B 0,C 180,E1 -27383.716,E2 -27383.716} C_VEL
LIN {X 0,Y 147.225,Z 597.655,A -85,B 0,C 180,E1 -27384.906,E2 -27384.906} C_VEL
LIN {X 0,Y 141.466,Z 611.039,A -85,B 0,C 180,E1 -27386.589,E2 -27386.589} C_VEL
LIN {X 0,Y 135.098,Z 623.397,A -85,B 0,C 180,E1 -27388.614,E2 -27388.614} C_VEL
LIN {X 0,Y 127.627,Z 635.962,A -85,B 0,C 180,E1 -27391.401,E2 -27391.401} C_VEL
LIN {X 0,Y 119.859,Z 647.382,A -85,B 0,C 180,E1 -27394.824,E2 -27394.824} C_VEL
LIN {X 0,Y 111.798,Z 657.903,A -85,B 0,C 180,E1 -27399.103,E2 -27399.103} C_VEL
LIN {X 0,Y 103.885,Z 667.65,A -85,B 0,C 180,E1 -27404.737,E2 -27404.737} C_VEL
LIN {X 0,Y 96.348,Z 676.227,A -85,B 0,C 180,E1 -27411.682,E2 -27411.682} C_VEL
LIN {X 0,Y 90.449,Z 683.105,A -85,B 0,C 180,E1 -27419.664,E2 -27419.664} C_VEL
LIN {X 0,Y 86.364,Z 688.489,A -85,B 0,C 180,E1 -27428.519,E2 -27428.519} C_VEL
LIN {X 0,Y 84.566,Z 691.58,A -85,B 0,C 180,E1 -27435.562,E2 -27435.562} C_VEL
LIN {X 0,Y 83.792,Z 694.629,A -85,B 0,C 180,E1 -27445.188,E2 -27445.188} C_VEL
LIN {X 0,Y 83.94,Z 695.688,A -85,B 0,C 180,E1 -27450,E2 -27450} C_VEL
LIN {X 0,Y 83.978,Z 696.861,A -85,B 0,C 180,E1 -27459.635,E2 -27459.635} C_VEL
LIN {X 0,Y 85.725,Z 696.849,A -85,B 0,C 180,E1 -27469.143,E2 -27469.143} C_VEL
LIN {X 0,Y 89.568,Z 695.74,A -85,B 0,C 180,E1 -27478.086,E2 -27478.086} C_VEL
LIN {X 0,Y 95.299,Z 693.523,A -85,B 0,C 180,E1 -27486.155,E2 -27486.155} C_VEL
LIN {X 0,Y 102.735,Z 690.156,A -85,B 0,C 180,E1 -27493.164,E2 -27493.164} C_VEL
LIN {X 0,Y 111.486,Z 685.518,A -85,B 0,C 180,E1 -27499.154,E2 -27499.154} C_VEL
LIN {X 0,Y 121.447,Z 679.363,A -85,B 0,C 180,E1 -27504.372,E2 -27504.372} C_VEL
LIN {X 0,Y 124.807,Z 676.811,A -85,B 0,C 180,E1 -27506.3,E2 -27506.3} C_VEL
LIN {X 0,Y 133.396,Z 668.706,A -85,B 0,C 180,E1 -27512.241,E2 -27512.241} C_VEL
LIN {X 0,Y 136.868,Z 665.614,A -85,B 0,C 180,E1 -27513.773,E2 -27513.773} C_VEL
LIN {X 0,Y 138.171,Z 664.491,A -85,B 0,C 180,E1 -27514.18,E2 -27514.18} C_VEL
LIN {X 0,Y 149.052,Z 654.77,A -85,B 0,C 180,E1 -27516.846,E2 -27516.846} C_VEL
LIN {X 0,Y 158.373,Z 645.154,A -85,B 0,C 180,E1 -27518.733,E2 -27518.733} C_VEL
LIN {X 0,Y 168.346,Z 632.986,A -85,B 0,C 180,E1 -27520.616,E2 -27520.616} C_VEL
LIN {X 0,Y 176.576,Z 621.307,A -85,B 0,C 180,E1 -27521.854,E2 -27521.854} C_VEL
LIN {X 0,Y 183.842,Z 609.073,A -85,B 0,C 180,E1 -27522.885,E2 -27522.885} C_VEL
LIN {X 0,Y 190.39,Z 595.817,A -85,B 0,C 180,E1 -27523.69,E2 -27523.69} C_VEL
LIN {X 0,Y 196.176,Z 581.245,A -85,B 0,C 180,E1 -27524.323,E2 -27524.323} C_VEL
LIN {X 0,Y 200.562,Z 566.626,A -85,B 0,C 180,E1 -27524.817,E2 -27524.817} C_VEL
LIN {X 0,Y 203.796,Z 551.21,A -85,B 0,C 180,E1 -27525.2,E2 -27525.2} C_VEL
LIN {X 0,Y 205.772,Z 535.785,A -85,B 0,C 180,E1 -27525.523,E2 -27525.523} C_VEL
LIN {X 0,Y 205.129,Z 533.618,A -85,B 0,C 180,E1 -27527.133,E2 -27527.133} C_VEL
LIN {X 0,Y 204.209,Z 531,A -85,B 0,C 180,E1 -27530.092,E2 -27530.092} C_VEL
LIN {X 0,Y 203.673,Z 528.453,A -85,B 0,C 180,E1 -27535.088,E2 -27535.088} C_VEL
LIN {X 0,Y 203.693,Z 528.675,A -85,B 0,C 180,E1 -27536.415,E2 -27536.415} C_VEL
LIN {X 0,Y 204.482,Z 531.528,A -85,B 0,C 180,E1 -27541.324,E2 -27541.324} C_VEL
LIN {X 0,Y 205.65,Z 534.985,A -85,B 0,C 180,E1 -27544.576,E2 -27544.576} C_VEL
LIN {X 0,Y 205.756,Z 535.295,A -85,B 0,C 180,E1 -27544.815,E2 -27544.815} C_VEL
LIN {X 0,Y 203.37,Z 552.34,A -85,B 0,C 180,E1 -27545.191,E2 -27545.191} C_VEL
LIN {X 0,Y 199.815,Z 568.007,A -85,B 0,C 180,E1 -27545.715,E2 -27545.715} C_VEL
LIN {X 0,Y 195.531,Z 581.44,A -85,B 0,C 180,E1 -27546.249,E2 -27546.249} C_VEL
LIN {X 0,Y 189.465,Z 596.293,A -85,B 0,C 180,E1 -27547.133,E2 -27547.133} C_VEL
LIN {X 0,Y 182.78,Z 609.331,A -85,B 0,C 180,E1 -27548.067,E2 -27548.067} C_VEL
LIN {X 0,Y 174.901,Z 622.164,A -85,B 0,C 180,E1 -27549.378,E2 -27549.378} C_VEL
LIN {X 0,Y 166.397,Z 633.784,A -85,B 0,C 180,E1 -27550.89,E2 -27550.89} C_VEL
LIN {X 0,Y 156.414,Z 645.324,A -85,B 0,C 180,E1 -27552.883,E2 -27552.883} C_VEL
LIN {X 0,Y 147.306,Z 654.393,A -85,B 0,C 180,E1 -27554.954,E2 -27554.954} C_VEL
LIN {X 0,Y 137.222,Z 663.045,A -85,B 0,C 180,E1 -27557.647,E2 -27557.647} C_VEL
LIN {X 0,Y 127.73,Z 670.115,A -85,B 0,C 180,E1 -27560.711,E2 -27560.711} C_VEL
LIN {X 0,Y 116.477,Z 677.338,A -85,B 0,C 180,E1 -27565.167,E2 -27565.167} C_VEL
LIN {X 0,Y 106.094,Z 682.976,A -85,B 0,C 180,E1 -27570.553,E2 -27570.553} C_VEL
LIN {X 0,Y 96.784,Z 687.189,A -85,B 0,C 180,E1 -27576.987,E2 -27576.987} C_VEL
LIN {X 0,Y 88.902,Z 690.097,A -85,B 0,C 180,E1 -27584.645,E2 -27584.645} C_VEL
LIN {X 0,Y 82.755,Z 691.78,A -85,B 0,C 180,E1 -27593.525,E2 -27593.525} C_VEL
LIN {X 0,Y 78.693,Z 692.278,A -85,B 0,C 180,E1 -27603.478,E2 -27603.478} C_VEL
LIN {X 0,Y 76.614,Z 691.58,A -85,B 0,C 180,E1 -27614.026,E2 -27614.026} C_VEL
LIN {X 0,Y 76.606,Z 689.709,A -85,B 0,C 180,E1 -27624.736,E2 -27624.736} C_VEL
LIN {X 0,Y 77.331,Z 688.336,A -85,B 0,C 180,E1 -27630,E2 -27630} C_VEL
LIN {X 0,Y 79.56,Z 684.723,A -85,B 0,C 180,E1 -27640.176,E2 -27640.176} C_VEL
LIN {X 0,Y 83.723,Z 679.842,A -85,B 0,C 180,E1 -27649.62,E2 -27649.62} C_VEL
LIN {X 0,Y 89.75,Z 673.559,A -85,B 0,C 180,E1 -27658.024,E2 -27658.024} C_VEL
LIN {X 0,Y 97.252,Z 665.691,A -85,B 0,C 180,E1 -27665.319,E2 -27665.319} C_VEL
LIN {X 0,Y 104.854,Z 657.311,A -85,B 0,C 180,E1 -27670.807,E2 -27670.807} C_VEL
LIN {X 0,Y 113.245,Z 647.226,A -85,B 0,C 180,E1 -27675.537,E2 -27675.537} C_VEL
LIN {X 0,Y 120.967,Z 636.924,A -85,B 0,C 180,E1 -27679.05,E2 -27679.05} C_VEL
LIN {X 0,Y 129.025,Z 624.583,A -85,B 0,C 180,E1 -27682.169,E2 -27682.169} C_VEL
LIN {X 0,Y 136.007,Z 612.227,A -85,B 0,C 180,E1 -27684.475,E2 -27684.475} C_VEL
LIN {X 0,Y 142.372,Z 598.736,A -85,B 0,C 180,E1 -27686.41,E2 -27686.41} C_VEL
LIN {X 0,Y 147.773,Z 584.756,A -85,B 0,C 180,E1 -27687.904,E2 -27687.904} C_VEL
LIN {X 0,Y 152.168,Z 570.371,A -85,B 0,C 180,E1 -27689.018,E2 -27689.018} C_VEL
LIN {X 0,Y 155.677,Z 554.496,A -85,B 0,C 180,E1 -27689.906,E2 -27689.906} C_VEL
LIN {X 0,Y 157.76,Z 539.89,A -85,B 0,C 180,E1 -27690.427,E2 -27690.427} C_VEL
LIN {X 0,Y 161.786,Z 500.241,A -85,B 0,C 180,E1 -27691.52,E2 -27691.52} C_VEL
LIN {X 0,Y 159.424,Z 494.28,A -85,B 0,C 180,E1 -27694.368,E2 -27694.368} C_VEL
LIN {X 0,Y 157.026,Z 488.832,A -85,B 0,C 180,E1 -27697.726,E2 -27697.726} C_VEL
LIN {X 0,Y 154.868,Z 484.185,A -85,B 0,C 180,E1 -27701.477,E2 -27701.477} C_VEL
LIN {X 0,Y 153.325,Z 480.978,A -85,B 0,C 180,E1 -27705.057,E2 -27705.057} C_VEL
LIN {X 0,Y 151.948,Z 477.414,A -85,B 0,C 180,E1 -27710.821,E2 -27710.821} C_VEL
LIN {X 0,Y 152.071,Z 477.276,A -85,B 0,C 180,E1 -27719.337,E2 -27719.337} C_VEL
LIN {X 0,Y 153.699,Z 481.517,A -85,B 0,C 180,E1 -27725.463,E2 -27725.463} C_VEL
LIN {X 0,Y 155.606,Z 485.706,A -85,B 0,C 180,E1 -27729.504,E2 -27729.504} C_VEL
LIN {X 0,Y 157.765,Z 490.306,A -85,B 0,C 180,E1 -27732.95,E2 -27732.95} C_VEL
LIN {X 0,Y 160.563,Z 496.956,A -85,B 0,C 180,E1 -27736.633,E2 -27736.633} C_VEL
LIN {X 0,Y 161.751,Z 500.98,A -85,B 0,C 180,E1 -27738.129,E2 -27738.129} C_VEL
LIN {X 0,Y 158.066,Z 537.906,A -85,B 0,C 180,E1 -27739.191,E2 -27739.191} C_VEL
LIN {X 0,Y 155.868,Z 555.326,A -85,B 0,C 180,E1 -27739.738,E2 -27739.738} C_VEL
LIN {X 0,Y 152.607,Z 570.887,A -85,B 0,C 180,E1 -27740.464,E2 -27740.464} C_VEL
LIN {X 0,Y 148.187,Z 585.843,A -85,B 0,C 180,E1 -27741.448,E2 -27741.448} C_VEL
LIN {X 0,Y 142.839,Z 599.831,A -85,B 0,C 180,E1 -27742.698,E2 -27742.698} C_VEL
LIN {X 0,Y 136.88,Z 612.887,A -85,B 0,C 180,E1 -27744.382,E2 -27744.382} C_VEL
LIN {X 0,Y 130.382,Z 624.807,A -85,B 0,C 180,E1 -27746.344,E2 -27746.344} C_VEL
LIN {X 0,Y 123.337,Z 636.095,A -85,B 0,C 180,E1 -27748.824,E2 -27748.824} C_VEL
LIN {X 0,Y 114.575,Z 648.296,A -85,B 0,C 180,E1 -27752.496,E2 -27752.496} C_VEL
LIN {X 0,Y 106.711,Z 658.018,A -85,B 0,C 180,E1 -27756.505,E2 -27756.505} C_VEL
LIN {X 0,Y 98.96,Z 667.029,A -85,B 0,C 180,E1 -27761.78,E2 -27761.78} C_VEL
LIN {X 0,Y 91.73,Z 674.688,A -85,B 0,C 180,E1 -27767.902,E2 -27767.902} C_VEL
LIN {X 0,Y 85.786,Z 681.017,A -85,B 0,C 180,E1 -27775.007,E2 -27775.007} C_VEL
LIN {X 0,Y 80.692,Z 686.812,A -85,B 0,C 180,E1 -27784.184,E2 -27784.184} C_VEL
LIN {X 0,Y 77.644,Z 691.21,A -85,B 0,C 180,E1 -27794.243,E2 -27794.243} C_VEL
LIN {X 0,Y 76.697,Z 694.316,A -85,B 0,C 180,E1 -27804.742,E2 -27804.742} C_VEL
LIN {X 0,Y 76.845,Z 695.403,A -85,B 0,C 180,E1 -27810,E2 -27810} C_VEL
LIN {X 0,Y 76.716,Z 696.161,A -85,B 0,C 180,E1 -27815.256,E2 -27815.256} C_VEL
LIN {X 0,Y 77.7,Z 696.76,A -85,B 0,C 180,E1 -27825.744,E2 -27825.744} C_VEL
LIN {X 0,Y 80.902,Z 696.251,A -85,B 0,C 180,E1 -27835.744,E2 -27835.744} C_VEL
LIN {X 0,Y 86.21,Z 694.644,A -85,B 0,C 180,E1 -27844.796,E2 -27844.796} C_VEL
LIN {X 0,Y 93.487,Z 691.916,A -85,B 0,C 180,E1 -27852.577,E2 -27852.577} C_VEL
LIN {X 0,Y 102.098,Z 687.962,A -85,B 0,C 180,E1 -27859.217,E2 -27859.217} C_VEL
LIN {X 0,Y 111.991,Z 682.71,A -85,B 0,C 180,E1 -27864.668,E2 -27864.668} C_VEL
LIN {X 0,Y 119.855,Z 677.865,A -85,B 0,C 180,E1 -27868.239,E2 -27868.239} C_VEL
LIN {X 0,Y 131.157,Z 670.034,A -85,B 0,C 180,E1 -27872.147,E2 -27872.147} C_VEL
LIN {X 0,Y 138.171,Z 664.491,A -85,B 0,C 180,E1 -27874.18,E2 -27874.18} C_VEL
LIN {X 0,Y 141.866,Z 661.154,A -85,B 0,C 180,E1 -27875.48,E2 -27875.48} C_VEL
LIN {X 0,Y 151.189,Z 650.796,A -85,B 0,C 180,E1 -27879.85,E2 -27879.85} C_VEL
LIN {X 0,Y 154.652,Z 646.963,A -85,B 0,C 180,E1 -27880.902,E2 -27880.902} C_VEL
LIN {X 0,Y 155.909,Z 645.584,A -85,B 0,C 180,E1 -27881.152,E2 -27881.152} C_VEL
LIN {X 0,Y 165.522,Z 634.314,A -85,B 0,C 180,E1 -27882.808,E2 -27882.808} C_VEL
LIN {X 0,Y 174.508,Z 621.972,A -85,B 0,C 180,E1 -27884.055,E2 -27884.055} C_VEL
LIN {X 0,Y 182.716,Z 608.368,A -85,B 0,C 180,E1 -27885.108,E2 -27885.108} C_VEL
LIN {X 0,Y 189.359,Z 595.033,A -85,B 0,C 180,E1 -27885.841,E2 -27885.841} C_VEL
LIN {X 0,Y 195.227,Z 580.289,A -85,B 0,C 180,E1 -27886.404,E2 -27886.404} C_VEL
LIN {X 0,Y 199.748,Z 565.124,A -85,B 0,C 180,E1 -27886.868,E2 -27886.868} C_VEL
LIN {X 0,Y 202.886,Z 549.85,A -85,B 0,C 180,E1 -27887.217,E2 -27887.217} C_VEL
LIN {X 0,Y 204.123,Z 540.652,A -85,B 0,C 180,E1 -27887.387,E2 -27887.387} C_VEL
LIN {X 0,Y 203.214,Z 537.885,A -85,B 0,C 180,E1 -27890.546,E2 -27890.546} C_VEL
LIN {X 0,Y 202.787,Z 535.637,A -85,B 0,C 180,E1 -27895.03,E2 -27895.03} C_VEL
LIN {X 0,Y 202.807,Z 535.763,A -85,B 0,C 180,E1 -27896.275,E2 -27896.275} C_VEL
LIN {X 0,Y 203.46,Z 538.396,A -85,B 0,C 180,E1 -27900.867,E2 -27900.867} C_VEL
LIN {X 0,Y 204.085,Z 540.495,A -85,B 0,C 180,E1 -27902.963,E2 -27902.963} C_VEL
LIN {X 0,Y 201.712,Z 555.421,A -85,B 0,C 180,E1 -27903.302,E2 -27903.302} C_VEL
LIN {X 0,Y 198.055,Z 570.218,A -85,B 0,C 180,E1 -27903.758,E2 -27903.758} C_VEL
LIN {X 0,Y 193.416,Z 583.958,A -85,B 0,C 180,E1 -27904.312,E2 -27904.312} C_VEL
LIN {X 0,Y 187.849,Z 597.027,A -85,B 0,C 180,E1 -27905.047,E2 -27905.047} C_VEL
LIN {X 0,Y 181.898,Z 608.506,A -85,B 0,C 180,E1 -27905.787,E2 -27905.787} C_VEL
LIN {X 0,Y 174.159,Z 621.097,A -85,B 0,C 180,E1 -27906.954,E2 -27906.954} C_VEL
LIN {X 0,Y 165.175,Z 633.294,A -85,B 0,C 180,E1 -27908.405,E2 -27908.405} C_VEL
LIN {X 0,Y 155.724,Z 644.157,A -85,B 0,C 180,E1 -27910.097,E2 -27910.097} C_VEL
LIN {X 0,Y 145.588,Z 654.083,A -85,B 0,C 180,E1 -27912.168,E2 -27912.168} C_VEL
LIN {X 0,Y 134.707,Z 663.181,A -85,B 0,C 180,E1 -27914.799,E2 -27914.799} C_VEL
LIN {X 0,Y 123.81,Z 670.977,A -85,B 0,C 180,E1 -27918.047,E2 -27918.047} C_VEL
LIN {X 0,Y 113.542,Z 677.254,A -85,B 0,C 180,E1 -27921.803,E2 -27921.803} C_VEL
LIN {X 0,Y 102.538,Z 682.964,A -85,B 0,C 180,E1 -27926.998,E2 -27926.998} C_VEL
LIN {X 0,Y 92.533,Z 687.244,A -85,B 0,C 180,E1 -27933.336,E2 -27933.336} C_VEL
LIN {X 0,Y 83.869,Z 690.217,A -85,B 0,C 180,E1 -27941.047,E2 -27941.047} C_VEL
LIN {X 0,Y 76.954,Z 691.961,A -85,B 0,C 180,E1 -27950.261,E2 -27950.261} C_VEL
LIN {X 0,Y 72.057,Z 692.501,A -85,B 0,C 180,E1 -27961.384,E2 -27961.384} C_VEL
LIN {X 0,Y 69.661,Z 691.849,A -85,B 0,C 180,E1 -27972.382,E2 -27972.382} C_VEL
LIN {X 0,Y 69.442,Z 690.036,A -85,B 0,C 180,E1 -27984.192,E2 -27984.192} C_VEL
LIN {X 0,Y 70.289,Z 688.507,A -85,B 0,C 180,E1 -27990.721,E2 -27990.721} C_VEL
LIN {X 0,Y 72.601,Z 685.138,A -85,B 0,C 180,E1 -28001.164,E2 -28001.164} C_VEL
LIN {X 0,Y 77.077,Z 680.324,A -85,B 0,C 180,E1 -28011.391,E2 -28011.391} C_VEL
LIN {X 0,Y 83.57,Z 674.111,A -85,B 0,C 180,E1 -28020.304,E2 -28020.304} C_VEL
LIN {X 0,Y 91.581,Z 666.32,A -85,B 0,C 180,E1 -28027.874,E2 -28027.874} C_VEL
LIN {X 0,Y 99.609,Z 658.028,A -85,B 0,C 180,E1 -28033.466,E2 -28033.466} C_VEL
LIN {X 0,Y 108.411,Z 648.044,A -85,B 0,C 180,E1 -28038.204,E2 -28038.204} C_VEL
LIN {X 0,Y 116.463,Z 637.848,A -85,B 0,C 180,E1 -28041.674,E2 -28041.674} C_VEL
LIN {X 0,Y 124.819,Z 625.663,A -85,B 0,C 180,E1 -28044.729,E2 -28044.729} C_VEL
LIN {X 0,Y 132.05,Z 613.446,A -85,B 0,C 180,E1 -28046.957,E2 -28046.957} C_VEL
LIN {X 0,Y 138.6,Z 600.168,A -85,B 0,C 180,E1 -28048.836,E2 -28048.836} C_VEL
LIN {X 0,Y 144.538,Z 585.473,A -85,B 0,C 180,E1 -28050.361,E2 -28050.361} C_VEL
LIN {X 0,Y 149.048,Z 571.217,A -85,B 0,C 180,E1 -28051.428,E2 -28051.428} C_VEL
LIN {X 0,Y 152.65,Z 555.728,A -85,B 0,C 180,E1 -28052.268,E2 -28052.268} C_VEL
LIN {X 0,Y 154.921,Z 540.563,A -85,B 0,C 180,E1 -28052.803,E2 -28052.803} C_VEL
LIN {X 0,Y 158.758,Z 503.682,A -85,B 0,C 180,E1 -28053.812,E2 -28053.812} C_VEL
LIN {X 0,Y 156.462,Z 497.752,A -85,B 0,C 180,E1 -28057.03,E2 -28057.03} C_VEL
LIN {X 0,Y 154.502,Z 493.083,A -85,B 0,C 180,E1 -28060.32,E2 -28060.32} C_VEL
LIN {X 0,Y 153.112,Z 489.95,A -85,B 0,C 180,E1 -28063.22,E2 -28063.22} C_VEL
LIN {X 0,Y 152.136,Z 487.712,A -85,B 0,C 180,E1 -28065.854,E2 -28065.854} C_VEL
LIN {X 0,Y 150.991,Z 484.406,A -85,B 0,C 180,E1 -28071.368,E2 -28071.368} C_VEL
LIN {X 0,Y 151.151,Z 484.291,A -85,B 0,C 180,E1 -28079.083,E2 -28079.083} C_VEL
LIN {X 0,Y 152.522,Z 488.302,A -85,B 0,C 180,E1 -28084.79,E2 -28084.79} C_VEL
LIN {X 0,Y 154.119,Z 492.13,A -85,B 0,C 180,E1 -28088.522,E2 -28088.522} C_VEL
LIN {X 0,Y 156.109,Z 496.735,A -85,B 0,C 180,E1 -28091.996,E2 -28091.996} C_VEL
LIN {X 0,Y 158.56,Z 503.034,A -85,B 0,C 180,E1 -28095.511,E2 -28095.511} C_VEL
LIN {X 0,Y 158.791,Z 504.333,A -85,B 0,C 180,E1 -28095.897,E2 -28095.897} C_VEL
LIN {X 0,Y 153.852,Z 550.233,A -85,B 0,C 180,E1 -28097.134,E2 -28097.134} C_VEL
LIN {X 0,Y 150.848,Z 566.328,A -85,B 0,C 180,E1 -28097.795,E2 -28097.795} C_VEL
LIN {X 0,Y 146.525,Z 581.844,A -85,B 0,C 180,E1 -28098.683,E2 -28098.683} C_VEL
LIN {X 0,Y 141.799,Z 594.723,A -85,B 0,C 180,E1 -28099.66,E2 -28099.66} C_VEL
LIN {X 0,Y 135.639,Z 608.545,A -85,B 0,C 180,E1 -28101.147,E2 -28101.147} C_VEL
LIN {X 0,Y 128.842,Z 621.232,A -85,B 0,C 180,E1 -28103.002,E2 -28103.002} C_VEL
LIN {X 0,Y 121.492,Z 633.008,A -85,B 0,C 180,E1 -28105.329,E2 -28105.329} C_VEL
LIN {X 0,Y 113.66,Z 643.936,A -85,B 0,C 180,E1 -28108.22,E2 -28108.22} C_VEL
LIN {X 0,Y 105.436,Z 654.066,A -85,B 0,C 180,E1 -28111.858,E2 -28111.858} C_VEL
LIN {X 0,Y 97.874,Z 662.618,A -85,B 0,C 180,E1 -28116.115,E2 -28116.115} C_VEL
LIN {X 0,Y 89.722,Z 671.01,A -85,B 0,C 180,E1 -28121.914,E2 -28121.914} C_VEL
LIN {X 0,Y 81.74,Z 678.866,A -85,B 0,C 180,E1 -28129.845,E2 -28129.845} C_VEL
LIN {X 0,Y 75.5,Z 685.088,A -85,B 0,C 180,E1 -28139.204,E2 -28139.204} C_VEL
LIN {X 0,Y 71.442,Z 689.865,A -85,B 0,C 180,E1 -28149.86,E2 -28149.86} C_VEL
LIN {X 0,Y 69.925,Z 692.58,A -85,B 0,C 180,E1 -28158.403,E2 -28158.403} C_VEL
LIN {X 0,Y 69.74,Z 695.117,A -85,B 0,C 180,E1 -28170,E2 -28170} C_VEL
LIN {X 0,Y 69.618,Z 695.881,A -85,B 0,C 180,E1 -28175.794,E2 -28175.794} C_VEL
LIN {X 0,Y 70.836,Z 696.526,A -85,B 0,C 180,E1 -28187.316,E2 -28187.316} C_VEL
LIN {X 0,Y 74.515,Z 696.07,A -85,B 0,C 180,E1 -28198.137,E2 -28198.137} C_VEL
LIN {X 0,Y 81.464,Z 694.161,A -85,B 0,C 180,E1 -28209.067,E2 -28209.067} C_VEL
LIN {X 0,Y 88.348,Z 691.836,A -85,B 0,C 180,E1 -28215.72,E2 -28215.72} C_VEL
LIN {X 0,Y 97.574,Z 687.918,A -85,B 0,C 180,E1 -28222.401,E2 -28222.401} C_VEL
LIN {X 0,Y 108,Z 682.726,A -85,B 0,C 180,E1 -28227.775,E2 -28227.775} C_VEL
LIN {X 0,Y 116.257,Z 677.947,A -85,B 0,C 180,E1 -28231.226,E2 -28231.226} C_VEL
LIN {X 0,Y 127.984,Z 670.185,A -85,B 0,C 180,E1 -28234.967,E2 -28234.967} C_VEL
LIN {X 0,Y 138.632,Z 661.965,A -85,B 0,C 180,E1 -28237.697,E2 -28237.697} C_VEL
LIN {X 0,Y 149.575,Z 652.094,A -85,B 0,C 180,E1 -28240.006,E2 -28240.006} C_VEL
LIN {X 0,Y 155.909,Z 645.584,A -85,B 0,C 180,E1 -28241.152,E2 -28241.152} C_VEL
LIN {X 0,Y 158.204,Z 642.885,A -85,B 0,C 180,E1 -28241.831,E2 -28241.831} C_VEL
LIN {X 0,Y 163.932,Z 634.497,A -85,B 0,C 180,E1 -28245.029,E2 -28245.029} C_VEL
LIN {X 0,Y 166.11,Z 631.539,A -85,B 0,C 180,E1 -28245.547,E2 -28245.547} C_VEL
LIN {X 0,Y 175.209,Z 618.786,A -85,B 0,C 180,E1 -28246.586,E2 -28246.586} C_VEL
LIN {X 0,Y 182.709,Z 606.091,A -85,B 0,C 180,E1 -28247.439,E2 -28247.439} C_VEL
LIN {X 0,Y 189.451,Z 592.237,A -85,B 0,C 180,E1 -28248.076,E2 -28248.076} C_VEL
LIN {X 0,Y 195.243,Z 577.108,A -85,B 0,C 180,E1 -28248.58,E2 -28248.58} C_VEL
LIN {X 0,Y 199.598,Z 561.725,A -85,B 0,C 180,E1 -28248.956,E2 -28248.956} C_VEL
LIN {X 0,Y 202.515,Z 546.155,A -85,B 0,C 180,E1 -28249.3,E2 -28249.3} C_VEL
LIN {X 0,Y 202.172,Z 544.756,A -85,B 0,C 180,E1 -28251.001,E2 -28251.001} C_VEL
LIN {X 0,Y 201.877,Z 542.793,A -85,B 0,C 180,E1 -28255.008,E2 -28255.008} C_VEL
LIN {X 0,Y 201.892,Z 542.896,A -85,B 0,C 180,E1 -28256.259,E2 -28256.259} C_VEL
LIN {X 0,Y 202.357,Z 545.24,A -85,B 0,C 180,E1 -28260.411,E2 -28260.411} C_VEL
LIN {X 0,Y 202.479,Z 545.842,A -85,B 0,C 180,E1 -28261.026,E2 -28261.026} C_VEL
LIN {X 0,Y 199.488,Z 561.438,A -85,B 0,C 180,E1 -28261.464,E2 -28261.464} C_VEL
LIN {X 0,Y 195.132,Z 576.54,A -85,B 0,C 180,E1 -28261.901,E2 -28261.901} C_VEL
LIN {X 0,Y 189.942,Z 590.185,A -85,B 0,C 180,E1 -28262.534,E2 -28262.534} C_VEL
LIN {X 0,Y 183.031,Z 604.491,A -85,B 0,C 180,E1 -28263.294,E2 -28263.294} C_VEL
LIN {X 0,Y 176.166,Z 616.206,A -85,B 0,C 180,E1 -28264.166,E2 -28264.166} C_VEL
LIN {X 0,Y 167.649,Z 628.429,A -85,B 0,C 180,E1 -28265.365,E2 -28265.365} C_VEL
LIN {X 0,Y 159.204,Z 638.754,A -85,B 0,C 180,E1 -28266.659,E2 -28266.659} C_VEL
LIN {X 0,Y 149.179,Z 649.187,A -85,B 0,C 180,E1 -28268.374,E2 -28268.374} C_VEL
LIN {X 0,Y 137.666,Z 659.344,A -85,B 0,C 180,E1 -28270.663,E2 -28270.663} C_VEL
LIN {X 0,Y 126.449,Z 667.723,A -85,B 0,C 180,E1 -28273.432,E2 -28273.432} C_VEL
LIN {X 0,Y 114.041,Z 675.536,A -85,B 0,C 180,E1 -28277.212,E2 -28277.212} C_VEL
LIN {X 0,Y 102.246,Z 681.691,A -85,B 0,C 180,E1 -28281.884,E2 -28281.884} C_VEL
LIN {X 0,Y 91.844,Z 686.132,A -85,B 0,C 180,E1 -28287.333,E2 -28287.333} C_VEL
LIN {X 0,Y 83.77,Z 688.976,A -85,B 0,C 180,E1 -28292.97,E2 -28292.97} C_VEL
LIN {X 0,Y 75.12,Z 691.388,A -85,B 0,C 180,E1 -28301.543,E2 -28301.543} C_VEL
LIN {X 0,Y 68.362,Z 692.588,A -85,B 0,C 180,E1 -28311.915,E2 -28311.915} C_VEL
LIN {X 0,Y 64.027,Z 692.564,A -85,B 0,C 180,E1 -28323.956,E2 -28323.956} C_VEL
LIN {X 0,Y 62.213,Z 691.384,A -85,B 0,C 180,E1 -28336.943,E2 -28336.943} C_VEL
LIN {X 0,Y 63.02,Z 689.048,A -85,B 0,C 180,E1 -28350,E2 -28350} C_VEL
LIN {X 0,Y 65.646,Z 685.555,A -85,B 0,C 180,E1 -28362.364,E2 -28362.364} C_VEL
LIN {X 0,Y 70.521,Z 680.806,A -85,B 0,C 180,E1 -28373.493,E2 -28373.493} C_VEL
LIN {X 0,Y 77.546,Z 674.662,A -85,B 0,C 180,E1 -28382.942,E2 -28382.942} C_VEL
LIN {X 0,Y 86.117,Z 666.949,A -85,B 0,C 180,E1 -28390.76,E2 -28390.76} C_VEL
LIN {X 0,Y 94.604,Z 658.741,A -85,B 0,C 180,E1 -28396.413,E2 -28396.413} C_VEL
LIN {X 0,Y 103.835,Z 648.858,A -85,B 0,C 180,E1 -28401.112,E2 -28401.112} C_VEL
LIN {X 0,Y 112.223,Z 638.729,A -85,B 0,C 180,E1 -28404.502,E2 -28404.502} C_VEL
LIN {X 0,Y 120.881,Z 626.688,A -85,B 0,C 180,E1 -28407.462,E2 -28407.462} C_VEL
LIN {X 0,Y 128.335,Z 614.617,A -85,B 0,C 180,E1 -28409.601,E2 -28409.601} C_VEL
LIN {X 0,Y 135.108,Z 601.541,A -85,B 0,C 180,E1 -28411.378,E2 -28411.378} C_VEL
LIN {X 0,Y 140.449,Z 589.112,A -85,B 0,C 180,E1 -28412.649,E2 -28412.649} C_VEL
LIN {X 0,Y 145.432,Z 574.632,A -85,B 0,C 180,E1 -28413.772,E2 -28413.772} C_VEL
LIN {X 0,Y 149.371,Z 559.294,A -85,B 0,C 180,E1 -28414.619,E2 -28414.619} C_VEL
LIN {X 0,Y 152.058,Z 543.537,A -85,B 0,C 180,E1 -28415.201,E2 -28415.201} C_VEL
LIN {X 0,Y 156.035,Z 507.505,A -85,B 0,C 180,E1 -28416.084,E2 -28416.084} C_VEL
LIN {X 0,Y 153.896,Z 501.697,A -85,B 0,C 180,E1 -28419.621,E2 -28419.621} C_VEL
LIN {X 0,Y 152.22,Z 497.461,A -85,B 0,C 180,E1 -28423.119,E2 -28423.119} C_VEL
LIN {X 0,Y 151.104,Z 494.654,A -85,B 0,C 180,E1 -28426.262,E2 -28426.262} C_VEL
LIN {X 0,Y 150.119,Z 491.508,A -85,B 0,C 180,E1 -28431.317,E2 -28431.317} C_VEL
LIN {X 0,Y 150.207,Z 491.28,A -85,B 0,C 180,E1 -28438.658,E2 -28438.658} C_VEL
LIN {X 0,Y 151.397,Z 495.162,A -85,B 0,C 180,E1 -28444.2,E2 -28444.2} C_VEL
LIN {X 0,Y 152.945,Z 499.195,A -85,B 0,C 180,E1 -28448.089,E2 -28448.089} C_VEL
LIN {X 0,Y 155.005,Z 504.514,A -85,B 0,C 180,E1 -28451.875,E2 -28451.875} C_VEL
LIN {X 0,Y 156.039,Z 507.446,A -85,B 0,C 180,E1 -28453.505,E2 -28453.505} C_VEL
LIN {X 0,Y 153.526,Z 531.565,A -85,B 0,C 180,E1 -28454.196,E2 -28454.196} C_VEL
LIN {X 0,Y 150.883,Z 552.929,A -85,B 0,C 180,E1 -28454.738,E2 -28454.738} C_VEL
LIN {X 0,Y 147.7,Z 568.339,A -85,B 0,C 180,E1 -28455.366,E2 -28455.366} C_VEL
LIN {X 0,Y 143.584,Z 582.402,A -85,B 0,C 180,E1 -28456.139,E2 -28456.139} C_VEL
LIN {X 0,Y 138.752,Z 595.187,A -85,B 0,C 180,E1 -28457.049,E2 -28457.049} C_VEL
LIN {X 0,Y 133.212,Z 607.264,A -85,B 0,C 180,E1 -28458.259,E2 -28458.259} C_VEL
LIN {X 0,Y 126.237,Z 620.161,A -85,B 0,C 180,E1 -28460.034,E2 -28460.034} C_VEL
LIN {X 0,Y 120.878,Z 628.762,A -85,B 0,C 180,E1 -28461.523,E2 -28461.523} C_VEL
LIN {X 0,Y 113.369,Z 639.312,A -85,B 0,C 180,E1 -28463.88,E2 -28463.88} C_VEL
LIN {X 0,Y 104.671,Z 650.073,A -85,B 0,C 180,E1 -28467.17,E2 -28467.17} C_VEL
LIN {X 0,Y 96.393,Z 659.185,A -85,B 0,C 180,E1 -28471.052,E2 -28471.052} C_VEL
LIN {X 0,Y 87.516,Z 668.144,A -85,B 0,C 180,E1 -28476.577,E2 -28476.577} C_VEL
LIN {X 0,Y 80.506,Z 674.596,A -85,B 0,C 180,E1 -28482.095,E2 -28482.095} C_VEL
LIN {X 0,Y 72.741,Z 681.586,A -85,B 0,C 180,E1 -28490.9,E2 -28490.9} C_VEL
LIN {X 0,Y 66.815,Z 687.222,A -85,B 0,C 180,E1 -28501.749,E2 -28501.749} C_VEL
LIN {X 0,Y 63.997,Z 690.472,A -85,B 0,C 180,E1 -28510.764,E2 -28510.764} C_VEL
LIN {X 0,Y 62.518,Z 693.691,A -85,B 0,C 180,E1 -28523.545,E2 -28523.545} C_VEL
LIN {X 0,Y 62.634,Z 694.817,A -85,B 0,C 180,E1 -28530,E2 -28530} C_VEL
LIN {X 0,Y 62.538,Z 695.595,A -85,B 0,C 180,E1 -28536.452,E2 -28536.452} C_VEL
LIN {X 0,Y 64.046,Z 696.292,A -85,B 0,C 180,E1 -28549.22,E2 -28549.22} C_VEL
LIN {X 0,Y 68.287,Z 695.889,A -85,B 0,C 180,E1 -28560.97,E2 -28560.97} C_VEL
LIN {X 0,Y 75.518,Z 694.186,A -85,B 0,C 180,E1 -28571.886,E2 -28571.886} C_VEL
LIN {X 0,Y 83.501,Z 691.742,A -85,B 0,C 180,E1 -28579.244,E2 -28579.244} C_VEL
LIN {X 0,Y 93.381,Z 687.874,A -85,B 0,C 180,E1 -28585.881,E2 -28585.881} C_VEL
LIN {X 0,Y 104.355,Z 682.745,A -85,B 0,C 180,E1 -28591.106,E2 -28591.106} C_VEL
LIN {X 0,Y 113.005,Z 678.034,A -85,B 0,C 180,E1 -28594.39,E2 -28594.39} C_VEL
LIN {X 0,Y 125.144,Z 670.349,A -85,B 0,C 180,E1 -28597.915,E2 -28597.915} C_VEL
LIN {X 0,Y 136.088,Z 662.176,A -85,B 0,C 180,E1 -28600.473,E2 -28600.473} C_VEL
LIN {X 0,Y 147.302,Z 652.387,A -85,B 0,C 180,E1 -28602.598,E2 -28602.598} C_VEL
LIN {X 0,Y 156.899,Z 642.571,A -85,B 0,C 180,E1 -28604.143,E2 -28604.143} C_VEL
LIN {X 0,Y 166.11,Z 631.539,A -85,B 0,C 180,E1 -28605.547,E2 -28605.547} C_VEL
LIN {X 0,Y 169.462,Z 627.024,A -85,B 0,C 180,E1 -28606.154,E2 -28606.154} C_VEL
LIN {X 0,Y 174.2,Z 619.601,A -85,B 0,C 180,E1 -28607.704,E2 -28607.704} C_VEL
LIN {X 0,Y 178.608,Z 611.886,A -85,B 0,C 180,E1 -28609.148,E2 -28609.148} C_VEL
LIN {X 0,Y 181.355,Z 606.866,A -85,B 0,C 180,E1 -28609.614,E2 -28609.614} C_VEL
LIN {X 0,Y 188.123,Z 593.373,A -85,B 0,C 180,E1 -28610.174,E2 -28610.174} C_VEL
LIN {X 0,Y 193.926,Z 578.805,A -85,B 0,C 180,E1 -28610.615,E2 -28610.615} C_VEL
LIN {X 0,Y 198.355,Z 564.084,A -85,B 0,C 180,E1 -28610.937,E2 -28610.937} C_VEL
LIN {X 0,Y 200.995,Z 551.698,A -85,B 0,C 180,E1 -28611.223,E2 -28611.223} C_VEL
LIN {X 0,Y 200.802,Z 549.893,A -85,B 0,C 180,E1 -28614.981,E2 -28614.981} C_VEL
LIN {X 0,Y 200.805,Z 549.99,A -85,B 0,C 180,E1 -28616.238,E2 -28616.238} C_VEL
LIN {X 0,Y 200.953,Z 551.476,A -85,B 0,C 180,E1 -28619.155,E2 -28619.155} C_VEL
LIN {X 0,Y 197.456,Z 566.843,A -85,B 0,C 180,E1 -28619.568,E2 -28619.568} C_VEL
LIN {X 0,Y 192.618,Z 581.746,A -85,B 0,C 180,E1 -28620.001,E2 -28620.001} C_VEL
LIN {X 0,Y 186.256,Z 596.694,A -85,B 0,C 180,E1 -28620.698,E2 -28620.698} C_VEL
LIN {X 0,Y 179.266,Z 609.775,A -85,B 0,C 180,E1 -28621.382,E2 -28621.382} C_VEL
LIN {X 0,Y 171.305,Z 622.163,A -85,B 0,C 180,E1 -28622.352,E2 -28622.352} C_VEL
LIN {X 0,Y 161.959,Z 634.299,A -85,B 0,C 180,E1 -28623.573,E2 -28623.573} C_VEL
LIN {X 0,Y 151.35,Z 645.832,A -85,B 0,C 180,E1 -28625.099,E2 -28625.099} C_VEL
LIN {X 0,Y 141.537,Z 654.942,A -85,B 0,C 180,E1 -28626.736,E2 -28626.736} C_VEL
LIN {X 0,Y 129.865,Z 664.128,A -85,B 0,C 180,E1 -28629.014,E2 -28629.014} C_VEL
LIN {X 0,Y 118.452,Z 671.707,A -85,B 0,C 180,E1 -28631.768,E2 -28631.768} C_VEL
LIN {X 0,Y 107.024,Z 678.108,A -85,B 0,C 180,E1 -28635.23,E2 -28635.23} C_VEL
LIN {X 0,Y 96.744,Z 682.952,A -85,B 0,C 180,E1 -28639.197,E2 -28639.197} C_VEL
LIN {X 0,Y 85.315,Z 687.361,A -85,B 0,C 180,E1 -28645.021,E2 -28645.021} C_VEL
LIN {X 0,Y 75.008,Z 690.457,A -85,B 0,C 180,E1 -28652.514,E2 -28652.514} C_VEL
LIN {X 0,Y 66.305,Z 692.313,A -85,B 0,C 180,E1 -28662.101,E2 -28662.101} C_VEL
LIN {X 0,Y 59.82,Z 692.933,A -85,B 0,C 180,E1 -28674.026,E2 -28674.026} C_VEL
LIN {X 0,Y 55.998,Z 692.386,A -85,B 0,C 180,E1 -28687.883,E2 -28687.883} C_VEL
LIN {X 0,Y 55.141,Z 690.69,A -85,B 0,C 180,E1 -28702.678,E2 -28702.678} C_VEL
LIN {X 0,Y 56.311,Z 688.762,A -85,B 0,C 180,E1 -28713.124,E2 -28713.124} C_VEL
LIN {X 0,Y 59.847,Z 684.906,A -85,B 0,C 180,E1 -28727.073,E2 -28727.073} C_VEL
LIN {X 0,Y 65.816,Z 679.868,A -85,B 0,C 180,E1 -28738.72,E2 -28738.72} C_VEL
LIN {X 0,Y 73.875,Z 673.415,A -85,B 0,C 180,E1 -28748.198,E2 -28748.198} C_VEL
LIN {X 0,Y 83.361,Z 665.362,A -85,B 0,C 180,E1 -28755.776,E2 -28755.776} C_VEL
LIN {X 0,Y 92.57,Z 656.773,A -85,B 0,C 180,E1 -28761.095,E2 -28761.095} C_VEL
LIN {X 0,Y 102.434,Z 646.442,A -85,B 0,C 180,E1 -28765.419,E2 -28765.419} C_VEL
LIN {X 0,Y 111.228,Z 635.857,A -85,B 0,C 180,E1 -28768.54,E2 -28768.54} C_VEL
LIN {X 0,Y 119.531,Z 624.324,A -85,B 0,C 180,E1 -28770.998,E2 -28770.998} C_VEL
LIN {X 0,Y 127.229,Z 611.771,A -85,B 0,C 180,E1 -28772.966,E2 -28772.966} C_VEL
LIN {X 0,Y 134.223,Z 598.001,A -85,B 0,C 180,E1 -28774.586,E2 -28774.586} C_VEL
LIN {X 0,Y 140.083,Z 583.646,A -85,B 0,C 180,E1 -28775.85,E2 -28775.85} C_VEL
LIN {X 0,Y 144.824,Z 568.691,A -85,B 0,C 180,E1 -28776.78,E2 -28776.78} C_VEL
LIN {X 0,Y 148.267,Z 553.659,A -85,B 0,C 180,E1 -28777.439,E2 -28777.439} C_VEL
LIN {X 0,Y 150.577,Z 537.696,A -85,B 0,C 180,E1 -28777.894,E2 -28777.894} C_VEL
LIN {X 0,Y 153.449,Z 511.703,A -85,B 0,C 180,E1 -28778.505,E2 -28778.505} C_VEL
LIN {X 0,Y 153.261,Z 510.7,A -85,B 0,C 180,E1 -28778.918,E2 -28778.918} C_VEL
LIN {X 0,Y 151.687,Z 506.144,A -85,B 0,C 180,E1 -28782.123,E2 -28782.123} C_VEL
LIN {X 0,Y 150.588,Z 503.181,A -85,B 0,C 180,E1 -28784.952,E2 -28784.952} C_VEL
LIN {X 0,Y 149.981,Z 501.379,A -85,B 0,C 180,E1 -28787.024,E2 -28787.024} C_VEL
LIN {X 0,Y 149.179,Z 498.467,A -85,B 0,C 180,E1 -28791.874,E2 -28791.874} C_VEL
LIN {X 0,Y 149.275,Z 498.353,A -85,B 0,C 180,E1 -28798.313,E2 -28798.313} C_VEL
LIN {X 0,Y 150.266,Z 501.935,A -85,B 0,C 180,E1 -28803.518,E2 -28803.518} C_VEL
LIN {X 0,Y 151.828,Z 506.385,A -85,B 0,C 180,E1 -28807.757,E2 -28807.757} C_VEL
LIN {X 0,Y 153.515,Z 511.367,A -85,B 0,C 180,E1 -28811.116,E2 -28811.116} C_VEL
LIN {X 0,Y 150.117,Z 542.353,A -85,B 0,C 180,E1 -28811.873,E2 -28811.873} C_VEL
LIN {X 0,Y 147.626,Z 558.546,A -85,B 0,C 180,E1 -28812.36,E2 -28812.36} C_VEL
LIN {X 0,Y 143.805,Z 574.016,A -85,B 0,C 180,E1 -28812.996,E2 -28812.996} C_VEL
LIN {X 0,Y 138.862,Z 588.585,A -85,B 0,C 180,E1 -28813.805,E2 -28813.805} C_VEL
LIN {X 0,Y 132.741,Z 602.753,A -85,B 0,C 180,E1 -28814.927,E2 -28814.927} C_VEL
LIN {X 0,Y 125.558,Z 616.46,A -85,B 0,C 180,E1 -28816.558,E2 -28816.558} C_VEL
LIN {X 0,Y 119.194,Z 626.555,A -85,B 0,C 180,E1 -28818.051,E2 -28818.051} C_VEL
LIN {X 0,Y 110.644,Z 638.434,A -85,B 0,C 180,E1 -28820.461,E2 -28820.461} C_VEL
LIN {X 0,Y 101.592,Z 649.309,A -85,B 0,C 180,E1 -28823.563,E2 -28823.563} C_VEL
LIN {X 0,Y 93.22,Z 658.163,A -85,B 0,C 180,E1 -28827.056,E2 -28827.056} C_VEL
LIN {X 0,Y 83.44,Z 667.551,A -85,B 0,C 180,E1 -28832.617,E2 -28832.617} C_VEL
LIN {X 0,Y 75.876,Z 674.038,A -85,B 0,C 180,E1 -28838.064,E2 -28838.064} C_VEL
LIN {X 0,Y 67.563,Z 680.893,A -85,B 0,C 180,E1 -28846.728,E2 -28846.728} C_VEL
LIN {X 0,Y 60.573,Z 686.793,A -85,B 0,C 180,E1 -28858.525,E2 -28858.525} C_VEL
LIN {X 0,Y 57.281,Z 690.102,A -85,B 0,C 180,E1 -28868.402,E2 -28868.402} C_VEL
LIN {X 0,Y 55.442,Z 693.367,A -85,B 0,C 180,E1 -28882.717,E2 -28882.717} C_VEL
LIN {X 0,Y 55.522,Z 694.507,A -85,B 0,C 180,E1 -28890,E2 -28890} C_VEL
LIN {X 0,Y 55.481,Z 695.31,A -85,B 0,C 180,E1 -28897.277,E2 -28897.277} C_VEL
LIN {X 0,Y 57.352,Z 696.058,A -85,B 0,C 180,E1 -28911.569,E2 -28911.569} C_VEL
LIN {X 0,Y 62.263,Z 695.708,A -85,B 0,C 180,E1 -28924.359,E2 -28924.359} C_VEL
LIN {X 0,Y 69.823,Z 694.202,A -85,B 0,C 180,E1 -28935.208,E2 -28935.208} C_VEL
LIN {X 0,Y 79.001,Z 691.643,A -85,B 0,C 180,E1 -28943.192,E2 -28943.192} C_VEL
LIN {X 0,Y 89.567,Z 687.837,A -85,B 0,C 180,E1 -28949.669,E2 -28949.669} C_VEL
LIN {X 0,Y 101.091,Z 682.771,A -85,B 0,C 180,E1 -28954.659,E2 -28954.659} C_VEL
LIN {X 0,Y 110.117,Z 678.108,A -85,B 0,C 180,E1 -28957.734,E2 -28957.734} C_VEL
LIN {X 0,Y 122.649,Z 670.496,A -85,B 0,C 180,E1 -28960.993,E2 -28960.993} C_VEL
LIN {X 0,Y 133.88,Z 662.379,A -85,B 0,C 180,E1 -28963.342,E2 -28963.342} C_VEL
LIN {X 0,Y 145.341,Z 652.677,A -85,B 0,C 180,E1 -28965.264,E2 -28965.264} C_VEL
LIN {X 0,Y 156.157,Z 641.846,A -85,B 0,C 180,E1 -28966.812,E2 -28966.812} C_VEL
LIN {X 0,Y 165.256,Z 631.092,A -85,B 0,C 180,E1 -28967.998,E2 -28967.998} C_VEL
LIN {X 0,Y 174.552,Z 618.168,A -85,B 0,C 180,E1 -28968.935,E2 -28968.935} C_VEL
LIN {X 0,Y 181.355,Z 606.866,A -85,B 0,C 180,E1 -28969.614,E2 -28969.614} C_VEL
LIN {X 0,Y 184.005,Z 601.835,A -85,B 0,C 180,E1 -28970.044,E2 -28970.044} C_VEL
LIN {X 0,Y 187.835,Z 593.461,A -85,B 0,C 180,E1 -28971.255,E2 -28971.255} C_VEL
LIN {X 0,Y 191.256,Z 584.941,A -85,B 0,C 180,E1 -28972.38,E2 -28972.38} C_VEL
LIN {X 0,Y 193.197,Z 579.477,A -85,B 0,C 180,E1 -28972.694,E2 -28972.694} C_VEL
LIN {X 0,Y 197.908,Z 564.096,A -85,B 0,C 180,E1 -28972.99,E2 -28972.99} C_VEL
LIN {X 0,Y 199.386,Z 557.856,A -85,B 0,C 180,E1 -28973.139,E2 -28973.139} C_VEL
LIN {X 0,Y 199.441,Z 556.914,A -85,B 0,C 180,E1 -28974.947,E2 -28974.947} C_VEL
LIN {X 0,Y 199.426,Z 557.057,A -85,B 0,C 180,E1 -28976.237,E2 -28976.237} C_VEL
LIN {X 0,Y 199.385,Z 557.587,A -85,B 0,C 180,E1 -28977.242,E2 -28977.242} C_VEL
LIN {X 0,Y 196.034,Z 570.477,A -85,B 0,C 180,E1 -28977.603,E2 -28977.603} C_VEL
LIN {X 0,Y 191.458,Z 583.688,A -85,B 0,C 180,E1 -28977.956,E2 -28977.956} C_VEL
LIN {X 0,Y 185.424,Z 597.427,A -85,B 0,C 180,E1 -28978.539,E2 -28978.539} C_VEL
LIN {X 0,Y 178.356,Z 610.409,A -85,B 0,C 180,E1 -28979.137,E2 -28979.137} C_VEL
LIN {X 0,Y 169.827,Z 623.343,A -85,B 0,C 180,E1 -28980.049,E2 -28980.049} C_VEL
LIN {X 0,Y 161.668,Z 633.806,A -85,B 0,C 180,E1 -28980.98,E2 -28980.98} C_VEL
LIN {X 0,Y 150.875,Z 645.457,A -85,B 0,C 180,E1 -28982.323,E2 -28982.323} C_VEL
LIN {X 0,Y 140.865,Z 654.629,A -85,B 0,C 180,E1 -28983.768,E2 -28983.768} C_VEL
LIN {X 0,Y 128.917,Z 663.904,A -85,B 0,C 180,E1 -28985.783,E2 -28985.783} C_VEL
LIN {X 0,Y 117.17,Z 671.56,A -85,B 0,C 180,E1 -28988.236,E2 -28988.236} C_VEL
LIN {X 0,Y 104.3,Z 678.555,A -85,B 0,C 180,E1 -28991.664,E2 -28991.664} C_VEL
LIN {X 0,Y 91.472,Z 684.199,A -85,B 0,C 180,E1 -28996.179,E2 -28996.179} C_VEL
LIN {X 0,Y 82.469,Z 687.422,A -85,B 0,C 180,E1 -29000.378,E2 -29000.378} C_VEL
LIN {X 0,Y 71.314,Z 690.58,A -85,B 0,C 180,E1 -29007.507,E2 -29007.507} C_VEL
LIN {X 0,Y 61.615,Z 692.47,A -85,B 0,C 180,E1 -29017.018,E2 -29017.018} C_VEL
LIN {X 0,Y 54.037,Z 693.145,A -85,B 0,C 180,E1 -29029.436,E2 -29029.436} C_VEL
LIN {X 0,Y 49.328,Z 692.655,A -85,B 0,C 180,E1 -29044.696,E2 -29044.696} C_VEL
LIN {X 0,Y 48,Z 691.016,A -85,B 0,C 180,E1 -29061.581,E2 -29061.581} C_VEL
LIN {X 0,Y 49.351,Z 688.948,A -85,B 0,C 180,E1 -29074.493,E2 -29074.493} C_VEL
LIN {X 0,Y 53.122,Z 685.319,A -85,B 0,C 180,E1 -29089.315,E2 -29089.315} C_VEL
LIN {X 0,Y 59.692,Z 680.347,A -85,B 0,C 180,E1 -29101.994,E2 -29101.994} C_VEL
LIN {X 0,Y 68.465,Z 673.961,A -85,B 0,C 180,E1 -29111.855,E2 -29111.855} C_VEL
LIN {X 0,Y 78.598,Z 665.982,A -85,B 0,C 180,E1 -29119.469,E2 -29119.469} C_VEL
LIN {X 0,Y 88.305,Z 657.476,A -85,B 0,C 180,E1 -29124.664,E2 -29124.664} C_VEL
LIN {X 0,Y 98.6,Z 647.239,A -85,B 0,C 180,E1 -29128.798,E2 -29128.798} C_VEL
LIN {X 0,Y 107.712,Z 636.768,A -85,B 0,C 180,E1 -29131.745,E2 -29131.745} C_VEL
LIN {X 0,Y 116.274,Z 625.374,A -85,B 0,C 180,E1 -29134.04,E2 -29134.04} C_VEL
LIN {X 0,Y 124.194,Z 612.994,A -85,B 0,C 180,E1 -29135.853,E2 -29135.853} C_VEL
LIN {X 0,Y 131.356,Z 599.47,A -85,B 0,C 180,E1 -29137.36,E2 -29137.36} C_VEL
LIN {X 0,Y 137.365,Z 585.454,A -85,B 0,C 180,E1 -29138.518,E2 -29138.518} C_VEL
LIN {X 0,Y 142.205,Z 571.032,A -85,B 0,C 180,E1 -29139.378,E2 -29139.378} C_VEL
LIN {X 0,Y 146.051,Z 555.22,A -85,B 0,C 180,E1 -29140.05,E2 -29140.05} C_VEL
LIN {X 0,Y 148.459,Z 539.675,A -85,B 0,C 180,E1 -29140.467,E2 -29140.467} C_VEL
LIN {X 0,Y 151.193,Z 515.442,A -85,B 0,C 180,E1 -29141.01,E2 -29141.01} C_VEL
LIN {X 0,Y 149.81,Z 510.953,A -85,B 0,C 180,E1 -29144.524,E2 -29144.524} C_VEL
LIN {X 0,Y 148.893,Z 508.192,A -85,B 0,C 180,E1 -29147.735,E2 -29147.735} C_VEL
LIN {X 0,Y 148.252,Z 505.481,A -85,B 0,C 180,E1 -29152.376,E2 -29152.376} C_VEL
LIN {X 0,Y 148.351,Z 505.401,A -85,B 0,C 180,E1 -29157.963,E2 -29157.963} C_VEL
LIN {X 0,Y 149.121,Z 508.633,A -85,B 0,C 180,E1 -29162.7,E2 -29162.7} C_VEL
LIN {X 0,Y 150.415,Z 512.765,A -85,B 0,C 180,E1 -29166.707,E2 -29166.707} C_VEL
LIN {X 0,Y 151.255,Z 515.474,A -85,B 0,C 180,E1 -29168.684,E2 -29168.684} C_VEL
LIN {X 0,Y 147.026,Z 550.866,A -85,B 0,C 180,E1 -29169.455,E2 -29169.455} C_VEL
LIN {X 0,Y 143.899,Z 566.144,A -85,B 0,C 180,E1 -29169.968,E2 -29169.968} C_VEL
LIN {X 0,Y 139.438,Z 581.144,A -85,B 0,C 180,E1 -29170.626,E2 -29170.626} C_VEL
LIN {X 0,Y 133.579,Z 595.969,A -85,B 0,C 180,E1 -29171.5,E2 -29171.5} C_VEL
LIN {X 0,Y 126.973,Z 609.428,A -85,B 0,C 180,E1 -29172.669,E2 -29172.669} C_VEL
LIN {X 0,Y 119.598,Z 621.872,A -85,B 0,C 180,E1 -29174.164,E2 -29174.164} C_VEL
LIN {X 0,Y 110.723,Z 634.508,A -85,B 0,C 180,E1 -29176.251,E2 -29176.251} C_VEL
LIN {X 0,Y 102.05,Z 645.087,A -85,B 0,C 180,E1 -29178.748,E2 -29178.748} C_VEL
LIN {X 0,Y 92.828,Z 654.875,A -85,B 0,C 180,E1 -29181.958,E2 -29181.958} C_VEL
LIN {X 0,Y 84.001,Z 663.224,A -85,B 0,C 180,E1 -29185.918,E2 -29185.918} C_VEL
LIN {X 0,Y 75.635,Z 670.357,A -85,B 0,C 180,E1 -29190.738,E2 -29190.738} C_VEL
LIN {X 0,Y 66.701,Z 677.294,A -85,B 0,C 180,E1 -29197.791,E2 -29197.791} C_VEL
LIN {X 0,Y 58.054,Z 683.712,A -85,B 0,C 180,E1 -29208.253,E2 -29208.253} C_VEL
LIN {X 0,Y 51.777,Z 688.669,A -85,B 0,C 180,E1 -29221.635,E2 -29221.635} C_VEL
LIN {X 0,Y 49.097,Z 691.548,A -85,B 0,C 180,E1 -29233.364,E2 -29233.364} C_VEL
LIN {X 0,Y 48.43,Z 694.195,A -85,B 0,C 180,E1 -29250,E2 -29250} C_VEL
LIN {X 0,Y 48.428,Z 695.024,A -85,B 0,C 180,E1 -29258.344,E2 -29258.344} C_VEL
LIN {X 0,Y 50.766,Z 695.824,A -85,B 0,C 180,E1 -29274.539,E2 -29274.539} C_VEL
LIN {X 0,Y 56.493,Z 695.528,A -85,B 0,C 180,E1 -29288.464,E2 -29288.464} C_VEL
LIN {X 0,Y 64.742,Z 694.126,A -85,B 0,C 180,E1 -29299.453,E2 -29299.453} C_VEL
LIN {X 0,Y 74.93,Z 691.548,A -85,B 0,C 180,E1 -29307.58,E2 -29307.58} C_VEL
LIN {X 0,Y 86.183,Z 687.8,A -85,B 0,C 180,E1 -29313.769,E2 -29313.769} C_VEL
LIN {X 0,Y 98.243,Z 682.797,A -85,B 0,C 180,E1 -29318.431,E2 -29318.431} C_VEL
LIN {X 0,Y 107.615,Z 678.168,A -85,B 0,C 180,E1 -29321.254,E2 -29321.254} C_VEL
LIN {X 0,Y 120.516,Z 670.625,A -85,B 0,C 180,E1 -29324.199,E2 -29324.199} C_VEL
LIN {X 0,Y 133.671,Z 661.352,A -85,B 0,C 180,E1 -29326.574,E2 -29326.574} C_VEL
LIN {X 0,Y 145.385,Z 651.486,A -85,B 0,C 180,E1 -29328.208,E2 -29328.208} C_VEL
LIN {X 0,Y 155.587,Z 641.3,A -85,B 0,C 180,E1 -29329.473,E2 -29329.473} C_VEL
LIN {X 0,Y 164.788,Z 630.541,A -85,B 0,C 180,E1 -29330.489,E2 -29330.489} C_VEL
LIN {X 0,Y 174.183,Z 617.555,A -85,B 0,C 180,E1 -29331.315,E2 -29331.315} C_VEL
LIN {X 0,Y 181.889,Z 604.672,A -85,B 0,C 180,E1 -29331.942,E2 -29331.942} C_VEL
LIN {X 0,Y 188.773,Z 590.569,A -85,B 0,C 180,E1 -29332.413,E2 -29332.413} C_VEL
LIN {X 0,Y 193.197,Z 579.477,A -85,B 0,C 180,E1 -29332.694,E2 -29332.694} C_VEL
LIN {X 0,Y 193.26,Z 579.169,A -85,B 0,C 180,E1 -29332.953,E2 -29332.953} C_VEL
LIN {X 0,Y 192.76,Z 580.301,A -85,B 0,C 180,E1 -29333.578,E2 -29333.578} C_VEL
LIN {X 0,Y 191.295,Z 583.891,A -85,B 0,C 180,E1 -29334.475,E2 -29334.475} C_VEL
LIN {X 0,Y 188.626,Z 590.128,A -85,B 0,C 180,E1 -29335.362,E2 -29335.362} C_VEL
LIN {X 0,Y 185.164,Z 597.594,A -85,B 0,C 180,E1 -29336.169,E2 -29336.169} C_VEL
LIN {X 0,Y 181.195,Z 605.09,A -85,B 0,C 180,E1 -29336.614,E2 -29336.614} C_VEL
LIN {X 0,Y 173.975,Z 616.933,A -85,B 0,C 180,E1 -29337.199,E2 -29337.199} C_VEL
LIN {X 0,Y 165.256,Z 628.927,A -85,B 0,C 180,E1 -29338.028,E2 -29338.028} C_VEL
LIN {X 0,Y 156.4,Z 639.273,A -85,B 0,C 180,E1 -29338.938,E2 -29338.938} C_VEL
LIN {X 0,Y 145.703,Z 649.844,A -85,B 0,C 180,E1 -29340.143,E2 -29340.143} C_VEL
LIN {X 0,Y 133.593,Z 659.903,A -85,B 0,C 180,E1 -29341.727,E2 -29341.727} C_VEL
LIN {X 0,Y 121.886,Z 668.034,A -85,B 0,C 180,E1 -29343.629,E2 -29343.629} C_VEL
LIN {X 0,Y 109.553,Z 675.215,A -85,B 0,C 180,E1 -29346.093,E2 -29346.093} C_VEL
LIN {X 0,Y 96.213,Z 681.583,A -85,B 0,C 180,E1 -29349.556,E2 -29349.556} C_VEL
LIN {X 0,Y 86.488,Z 685.388,A -85,B 0,C 180,E1 -29352.808,E2 -29352.808} C_VEL
LIN {X 0,Y 74.087,Z 689.252,A -85,B 0,C 180,E1 -29358.448,E2 -29358.448} C_VEL
LIN {X 0,Y 61.535,Z 692.01,A -85,B 0,C 180,E1 -29367.187,E2 -29367.187} C_VEL
LIN {X 0,Y 52.76,Z 693.138,A -85,B 0,C 180,E1 -29376.943,E2 -29376.943} C_VEL
LIN {X 0,Y 45.38,Z 693.283,A -85,B 0,C 180,E1 -29391.722,E2 -29391.722} C_VEL
LIN {X 0,Y 41.33,Z 692.277,A -85,B 0,C 180,E1 -29410.118,E2 -29410.118} C_VEL
LIN {X 0,Y 41.464,Z 690.115,A -85,B 0,C 180,E1 -29430.001,E2 -29430.001} C_VEL
LIN {X 0,Y 42.928,Z 688.599,A -85,B 0,C 180,E1 -29439.423,E2 -29439.423} C_VEL
LIN {X 0,Y 48.058,Z 684.663,A -85,B 0,C 180,E1 -29456.023,E2 -29456.023} C_VEL
LIN {X 0,Y 56.026,Z 679.402,A -85,B 0,C 180,E1 -29468.846,E2 -29468.846} C_VEL
LIN {X 0,Y 65.986,Z 672.701,A -85,B 0,C 180,E1 -29478.207,E2 -29478.207} C_VEL
LIN {X 0,Y 77.085,Z 664.373,A -85,B 0,C 180,E1 -29485.141,E2 -29485.141} C_VEL
LIN {X 0,Y 87.444,Z 655.481,A -85,B 0,C 180,E1 -29489.769,E2 -29489.769} C_VEL
LIN {X 0,Y 96.676,Z 646.42,A -85,B 0,C 180,E1 -29492.941,E2 -29492.941} C_VEL
LIN {X 0,Y 106.15,Z 635.737,A -85,B 0,C 180,E1 -29495.557,E2 -29495.557} C_VEL
LIN {X 0,Y 114.971,Z 624.095,A -85,B 0,C 180,E1 -29497.605,E2 -29497.605} C_VEL
LIN {X 0,Y 123.09,Z 611.401,A -85,B 0,C 180,E1 -29499.222,E2 -29499.222} C_VEL
LIN {X 0,Y 130.452,Z 597.43,A -85,B 0,C 180,E1 -29500.528,E2 -29500.528} C_VEL
LIN {X 0,Y 136.588,Z 582.797,A -85,B 0,C 180,E1 -29501.566,E2 -29501.566} C_VEL
LIN {X 0,Y 141.534,Z 567.393,A -85,B 0,C 180,E1 -29502.323,E2 -29502.323} C_VEL
LIN {X 0,Y 144.989,Z 552.216,A -85,B 0,C 180,E1 -29502.85,E2 -29502.85} C_VEL
LIN {X 0,Y 147.689,Z 532.639,A -85,B 0,C 180,E1 -29503.292,E2 -29503.292} C_VEL
LIN {X 0,Y 149.171,Z 519.716,A -85,B 0,C 180,E1 -29503.578,E2 -29503.578} C_VEL
LIN {X 0,Y 148.236,Z 516.482,A -85,B 0,C 180,E1 -29506.635,E2 -29506.635} C_VEL
LIN {X 0,Y 147.758,Z 514.785,A -85,B 0,C 180,E1 -29508.818,E2 -29508.818} C_VEL
LIN {X 0,Y 147.37,Z 512.539,A -85,B 0,C 180,E1 -29512.463,E2 -29512.463} C_VEL
LIN {X 0,Y 147.429,Z 512.408,A -85,B 0,C 180,E1 -29517.544,E2 -29517.544} C_VEL
LIN {X 0,Y 147.993,Z 515.226,A -85,B 0,C 180,E1 -29521.785,E2 -29521.785} C_VEL
LIN {X 0,Y 149.077,Z 519.276,A -85,B 0,C 180,E1 -29525.719,E2 -29525.719} C_VEL
LIN {X 0,Y 149.212,Z 519.786,A -85,B 0,C 180,E1 -29526.111,E2 -29526.111} C_VEL
LIN {X 0,Y 145.266,Z 551.545,A -85,B 0,C 180,E1 -29526.769,E2 -29526.769} C_VEL
LIN {X 0,Y 142.014,Z 566.774,A -85,B 0,C 180,E1 -29527.24,E2 -29527.24} C_VEL
LIN {X 0,Y 137.445,Z 581.641,A -85,B 0,C 180,E1 -29527.814,E2 -29527.814} C_VEL
LIN {X 0,Y 131.489,Z 596.31,A -85,B 0,C 180,E1 -29528.576,E2 -29528.576} C_VEL
LIN {X 0,Y 124.881,Z 609.453,A -85,B 0,C 180,E1 -29529.591,E2 -29529.591} C_VEL
LIN {X 0,Y 117.213,Z 622.062,A -85,B 0,C 180,E1 -29530.936,E2 -29530.936} C_VEL
LIN {X 0,Y 108.109,Z 634.627,A -85,B 0,C 180,E1 -29532.805,E2 -29532.805} C_VEL
LIN {X 0,Y 98.357,Z 646.057,A -85,B 0,C 180,E1 -29535.282,E2 -29535.282} C_VEL
LIN {X 0,Y 87.145,Z 657.202,A -85,B 0,C 180,E1 -29538.818,E2 -29538.818} C_VEL
LIN {X 0,Y 76.636,Z 666.332,A -85,B 0,C 180,E1 -29543.498,E2 -29543.498} C_VEL
LIN {X 0,Y 66.577,Z 673.932,A -85,B 0,C 180,E1 -29549.437,E2 -29549.437} C_VEL
LIN {X 0,Y 56.581,Z 680.817,A -85,B 0,C 180,E1 -29558.39,E2 -29558.39} C_VEL
LIN {X 0,Y 48.895,Z 685.928,A -85,B 0,C 180,E1 -29569.697,E2 -29569.697} C_VEL
LIN {X 0,Y 44.25,Z 689.347,A -85,B 0,C 180,E1 -29581.544,E2 -29581.544} C_VEL
LIN {X 0,Y 41.347,Z 692.688,A -85,B 0,C 180,E1 -29600.213,E2 -29600.213} C_VEL
LIN {X 0,Y 41.321,Z 693.881,A -85,B 0,C 180,E1 -29609.999,E2 -29609.999} C_VEL
LIN {X 0,Y 41.39,Z 694.737,A -85,B 0,C 180,E1 -29619.776,E2 -29619.776} C_VEL
LIN {X 0,Y 44.347,Z 695.589,A -85,B 0,C 180,E1 -29638.387,E2 -29638.387} C_VEL
LIN {X 0,Y 51.068,Z 695.348,A -85,B 0,C 180,E1 -29653.479,E2 -29653.479} C_VEL
LIN {X 0,Y 60.343,Z 693.978,A -85,B 0,C 180,E1 -29664.615,E2 -29664.615} C_VEL
LIN {X 0,Y 71.347,Z 691.453,A -85,B 0,C 180,E1 -29672.441,E2 -29672.441} C_VEL
LIN {X 0,Y 83.278,Z 687.764,A -85,B 0,C 180,E1 -29678.173,E2 -29678.173} C_VEL
LIN {X 0,Y 95.844,Z 682.822,A -85,B 0,C 180,E1 -29682.413,E2 -29682.413} C_VEL
LIN {X 0,Y 105.539,Z 678.226,A -85,B 0,C 180,E1 -29684.923,E2 -29684.923} C_VEL
LIN {X 0,Y 118.771,Z 670.752,A -85,B 0,C 180,E1 -29687.515,E2 -29687.515} C_VEL
LIN {X 0,Y 132.204,Z 661.56,A -85,B 0,C 180,E1 -29689.567,E2 -29689.567} C_VEL
LIN {X 0,Y 144.102,Z 651.778,A -85,B 0,C 180,E1 -29690.972,E2 -29690.972} C_VEL
LIN {X 0,Y 155.075,Z 641.045,A -85,B 0,C 180,E1 -29692.122,E2 -29692.122} C_VEL
LIN {X 0,Y 163.77,Z 631.053,A -85,B 0,C 180,E1 -29692.925,E2 -29692.925} C_VEL
LIN {X 0,Y 173.258,Z 618.219,A -85,B 0,C 180,E1 -29693.622,E2 -29693.622} C_VEL
LIN {X 0,Y 181.036,Z 605.534,A -85,B 0,C 180,E1 -29694.15,E2 -29694.15} C_VEL
LIN {X 0,Y 187.973,Z 591.707,A -85,B 0,C 180,E1 -29694.542,E2 -29694.542} C_VEL
LIN {X 0,Y 193.756,Z 577.097,A -85,B 0,C 180,E1 -29694.855,E2 -29694.855} C_VEL
LIN {X 0,Y 197.783,Z 563.826,A -85,B 0,C 180,E1 -29695.076,E2 -29695.076} C_VEL
LIN {X 0,Y 197.782,Z 563.81,A -85,B 0,C 180,E1 -29695.357,E2 -29695.357} C_VEL
LIN {X 0,Y 193.179,Z 578.747,A -85,B 0,C 180,E1 -29695.687,E2 -29695.687} C_VEL
LIN {X 0,Y 187.991,Z 591.565,A -85,B 0,C 180,E1 -29696.12,E2 -29696.12} C_VEL
LIN {X 0,Y 181.195,Z 605.09,A -85,B 0,C 180,E1 -29696.614,E2 -29696.614} C_VEL
LIN {X 0,Y 178.492,Z 609.804,A -85,B 0,C 180,E1 -29696.702,E2 -29696.702} C_VEL
LIN {X 0,Y 172.619,Z 618.935,A -85,B 0,C 180,E1 -29696.53,E2 -29696.53} C_VEL
LIN {X 0,Y 166.206,Z 627.678,A -85,B 0,C 180,E1 -29696.207,E2 -29696.207} C_VEL
LIN {X 0,Y 159.273,Z 635.951,A -85,B 0,C 180,E1 -29696.144,E2 -29696.144} C_VEL
LIN {X 0,Y 155.645,Z 639.906,A -85,B 0,C 180,E1 -29696.362,E2 -29696.362} C_VEL
LIN {X 0,Y 144.923,Z 650.348,A -85,B 0,C 180,E1 -29697.365,E2 -29697.365} C_VEL
LIN {X 0,Y 133.572,Z 659.631,A -85,B 0,C 180,E1 -29698.595,E2 -29698.595} C_VEL
LIN {X 0,Y 121.74,Z 667.786,A -85,B 0,C 180,E1 -29700.161,E2 -29700.161} C_VEL
LIN {X 0,Y 109.017,Z 675.106,A -85,B 0,C 180,E1 -29702.233,E2 -29702.233} C_VEL
LIN {X 0,Y 95.267,Z 681.546,A -85,B 0,C 180,E1 -29705.181,E2 -29705.181} C_VEL
LIN {X 0,Y 81.84,Z 686.486,A -85,B 0,C 180,E1 -29709.046,E2 -29709.046} C_VEL
LIN {X 0,Y 72.092,Z 689.33,A -85,B 0,C 180,E1 -29712.874,E2 -29712.874} C_VEL
LIN {X 0,Y 59.772,Z 691.933,A -85,B 0,C 180,E1 -29719.84,E2 -29719.84} C_VEL
LIN {X 0,Y 48.686,Z 693.321,A -85,B 0,C 180,E1 -29729.989,E2 -29729.989} C_VEL
LIN {X 0,Y 39.884,Z 693.524,A -85,B 0,C 180,E1 -29745.184,E2 -29745.184} C_VEL
LIN {X 0,Y 34.584,Z 692.573,A -85,B 0,C 180,E1 -29766.02,E2 -29766.02} C_VEL
LIN {X 0,Y 34.278,Z 690.467,A -85,B 0,C 180,E1 -29790.001,E2 -29790.001} C_VEL
LIN {X 0,Y 35.926,Z 688.976,A -85,B 0,C 180,E1 -29801.282,E2 -29801.282} C_VEL
LIN {X 0,Y 41.817,Z 685.072,A -85,B 0,C 180,E1 -29820.279,E2 -29820.279} C_VEL
LIN {X 0,Y 50.699,Z 679.874,A -85,B 0,C 180,E1 -29833.877,E2 -29833.877} C_VEL
LIN {X 0,Y 61.49,Z 673.241,A -85,B 0,C 180,E1 -29843.137,E2 -29843.137} C_VEL
LIN {X 0,Y 71.752,Z 666.1,A -85,B 0,C 180,E1 -29848.988,E2 -29848.988} C_VEL
LIN {X 0,Y 82.531,Z 657.526,A -85,B 0,C 180,E1 -29853.398,E2 -29853.398} C_VEL
LIN {X 0,Y 93.676,Z 647.215,A -85,B 0,C 180,E1 -29856.789,E2 -29856.789} C_VEL
LIN {X 0,Y 103.429,Z 636.647,A -85,B 0,C 180,E1 -29859.118,E2 -29859.118} C_VEL
LIN {X 0,Y 112.473,Z 625.145,A -85,B 0,C 180,E1 -29860.928,E2 -29860.928} C_VEL
LIN {X 0,Y 120.782,Z 612.622,A -85,B 0,C 180,E1 -29862.332,E2 -29862.332} C_VEL
LIN {X 0,Y 128.278,Z 598.899,A -85,B 0,C 180,E1 -29863.493,E2 -29863.493} C_VEL
LIN {X 0,Y 134.532,Z 584.611,A -85,B 0,C 180,E1 -29864.406,E2 -29864.406} C_VEL
LIN {X 0,Y 139.599,Z 569.621,A -85,B 0,C 180,E1 -29865.085,E2 -29865.085} C_VEL
LIN {X 0,Y 143.299,Z 554.456,A -85,B 0,C 180,E1 -29865.564,E2 -29865.564} C_VEL
LIN {X 0,Y 145.797,Z 538.205,A -85,B 0,C 180,E1 -29865.909,E2 -29865.909} C_VEL
LIN {X 0,Y 147.419,Z 524.301,A -85,B 0,C 180,E1 -29866.208,E2 -29866.208} C_VEL
LIN {X 0,Y 146.774,Z 521.703,A -85,B 0,C 180,E1 -29869.306,E2 -29869.306} C_VEL
LIN {X 0,Y 146.45,Z 519.532,A -85,B 0,C 180,E1 -29873.108,E2 -29873.108} C_VEL
LIN {X 0,Y 146.53,Z 519.564,A -85,B 0,C 180,E1 -29877.422,E2 -29877.422} C_VEL
LIN {X 0,Y 146.984,Z 522.302,A -85,B 0,C 180,E1 -29881.36,E2 -29881.36} C_VEL
LIN {X 0,Y 147.463,Z 524.432,A -85,B 0,C 180,E1 -29883.542,E2 -29883.542} C_VEL
LIN {X 0,Y 143.956,Z 551.551,A -85,B 0,C 180,E1 -29884.003,E2 -29884.003} C_VEL
LIN {X 0,Y 140.756,Z 566.325,A -85,B 0,C 180,E1 -29884.4,E2 -29884.4} C_VEL
LIN {X 0,Y 136.219,Z 580.982,A -85,B 0,C 180,E1 -29884.863,E2 -29884.863} C_VEL
LIN {X 0,Y 130.609,Z 594.836,A -85,B 0,C 180,E1 -29885.451,E2 -29885.451} C_VEL
LIN {X 0,Y 124.374,Z 607.244,A -85,B 0,C 180,E1 -29886.237,E2 -29886.237} C_VEL
LIN {X 0,Y 116.931,Z 619.652,A -85,B 0,C 180,E1 -29887.38,E2 -29887.38} C_VEL
LIN {X 0,Y 110.974,Z 628.207,A -85,B 0,C 180,E1 -29888.296,E2 -29888.296} C_VEL
LIN {X 0,Y 101.713,Z 639.705,A -85,B 0,C 180,E1 -29890.059,E2 -29890.059} C_VEL
LIN {X 0,Y 91.741,Z 650.261,A -85,B 0,C 180,E1 -29892.38,E2 -29892.38} C_VEL
LIN {X 0,Y 81.602,Z 659.499,A -85,B 0,C 180,E1 -29895.381,E2 -29895.381} C_VEL
LIN {X 0,Y 70.948,Z 668.003,A -85,B 0,C 180,E1 -29899.769,E2 -29899.769} C_VEL
LIN {X 0,Y 58.979,Z 676.219,A -85,B 0,C 180,E1 -29906.655,E2 -29906.655} C_VEL
LIN {X 0,Y 48.284,Z 682.775,A -85,B 0,C 180,E1 -29916.816,E2 -29916.816} C_VEL
LIN {X 0,Y 39.75,Z 687.86,A -85,B 0,C 180,E1 -29931.769,E2 -29931.769} C_VEL
LIN {X 0,Y 35.639,Z 690.804,A -85,B 0,C 180,E1 -29946.771,E2 -29946.771} C_VEL
LIN {X 0,Y 34.229,Z 693.566,A -85,B 0,C 180,E1 -29969.999,E2 -29969.999} C_VEL
LIN {X 0,Y 34.402,Z 694.449,A -85,B 0,C 180,E1 -29981.787,E2 -29981.787} C_VEL
LIN {X 0,Y 38.197,Z 695.355,A -85,B 0,C 180,E1 -30003.502,E2 -30003.502} C_VEL
LIN {X 0,Y 46.126,Z 695.169,A -85,B 0,C 180,E1 -30019.626,E2 -30019.626} C_VEL
LIN {X 0,Y 56.504,Z 693.827,A -85,B 0,C 180,E1 -30030.536,E2 -30030.536} C_VEL
LIN {X 0,Y 68.327,Z 691.358,A -85,B 0,C 180,E1 -30037.776,E2 -30037.776} C_VEL
LIN {X 0,Y 80.898,Z 687.727,A -85,B 0,C 180,E1 -30042.866,E2 -30042.866} C_VEL
LIN {X 0,Y 93.931,Z 682.848,A -85,B 0,C 180,E1 -30046.575,E2 -30046.575} C_VEL
LIN {X 0,Y 107.277,Z 676.591,A -85,B 0,C 180,E1 -30049.325,E2 -30049.325} C_VEL
LIN {X 0,Y 120.844,Z 668.781,A -85,B 0,C 180,E1 -30051.372,E2 -30051.372} C_VEL
LIN {X 0,Y 132.82,Z 660.508,A -85,B 0,C 180,E1 -30052.807,E2 -30052.807} C_VEL
LIN {X 0,Y 144.89,Z 650.565,A -85,B 0,C 180,E1 -30053.916,E2 -30053.916} C_VEL
LIN {X 0,Y 155.253,Z 640.423,A -85,B 0,C 180,E1 -30054.807,E2 -30054.807} C_VEL
LIN {X 0,Y 162.178,Z 632.632,A -85,B 0,C 180,E1 -30055.35,E2 -30055.35} C_VEL
LIN {X 0,Y 162.08,Z 632.727,A -85,B 0,C 180,E1 -30055.799,E2 -30055.799} C_VEL
LIN {X 0,Y 155.645,Z 639.906,A -85,B 0,C 180,E1 -30056.362,E2 -30056.362} C_VEL
LIN {X 0,Y 149.482,Z 646.113,A -85,B 0,C 180,E1 -30056.686,E2 -30056.686} C_VEL
LIN {X 0,Y 138.486,Z 655.853,A -85,B 0,C 180,E1 -30056.587,E2 -30056.587} C_VEL
LIN {X 0,Y 129.129,Z 662.937,A -85,B 0,C 180,E1 -30056.476,E2 -30056.476} C_VEL
LIN {X 0,Y 121.823,Z 667.744,A -85,B 0,C 180,E1 -30056.777,E2 -30056.777} C_VEL
LIN {X 0,Y 119.355,Z 669.227,A -85,B 0,C 180,E1 -30057.016,E2 -30057.016} C_VEL
LIN {X 0,Y 105.439,Z 676.818,A -85,B 0,C 180,E1 -30058.909,E2 -30058.909} C_VEL
LIN {X 0,Y 91.393,Z 682.936,A -85,B 0,C 180,E1 -30061.437,E2 -30061.437} C_VEL
LIN {X 0,Y 77.586,Z 687.583,A -85,B 0,C 180,E1 -30064.857,E2 -30064.857} C_VEL
LIN {X 0,Y 64.165,Z 690.88,A -85,B 0,C 180,E1 -30069.676,E2 -30069.676} C_VEL
LIN {X 0,Y 51.423,Z 692.929,A -85,B 0,C 180,E1 -30076.926,E2 -30076.926} C_VEL
LIN {X 0,Y 39.939,Z 693.781,A -85,B 0,C 180,E1 -30088.377,E2 -30088.377} C_VEL
LIN {X 0,Y 30.997,Z 693.461,A -85,B 0,C 180,E1 -30107.141,E2 -30107.141} C_VEL
LIN {X 0,Y 26.754,Z 691.99,A -85,B 0,C 180,E1 -30134.771,E2 -30134.771} C_VEL
LIN {X 0,Y 29,Z 689.337,A -85,B 0,C 180,E1 -30164.026,E2 -30164.026} C_VEL
LIN {X 0,Y 35.886,Z 685.48,A -85,B 0,C 180,E1 -30185.983,E2 -30185.983} C_VEL
LIN {X 0,Y 45.855,Z 680.346,A -85,B 0,C 180,E1 -30200.027,E2 -30200.027} C_VEL
LIN {X 0,Y 57.519,Z 673.782,A -85,B 0,C 180,E1 -30208.794,E2 -30208.794} C_VEL
LIN {X 0,Y 68.383,Z 666.713,A -85,B 0,C 180,E1 -30214.065,E2 -30214.065} C_VEL
LIN {X 0,Y 79.621,Z 658.224,A -85,B 0,C 180,E1 -30217.945,E2 -30217.945} C_VEL
LIN {X 0,Y 91.126,Z 648.01,A -85,B 0,C 180,E1 -30220.87,E2 -30220.87} C_VEL
LIN {X 0,Y 101.13,Z 637.558,A -85,B 0,C 180,E1 -30222.855,E2 -30222.855} C_VEL
LIN {X 0,Y 110.371,Z 626.194,A -85,B 0,C 180,E1 -30224.389,E2 -30224.389} C_VEL
LIN {X 0,Y 118.84,Z 613.845,A -85,B 0,C 180,E1 -30225.557,E2 -30225.557} C_VEL
LIN {X 0,Y 126.458,Z 600.366,A -85,B 0,C 180,E1 -30226.552,E2 -30226.552} C_VEL
LIN {X 0,Y 132.816,Z 586.411,A -85,B 0,C 180,E1 -30227.325,E2 -30227.325} C_VEL
LIN {X 0,Y 138.177,Z 571.213,A -85,B 0,C 180,E1 -30227.928,E2 -30227.928} C_VEL
LIN {X 0,Y 142.142,Z 555.605,A -85,B 0,C 180,E1 -30228.367,E2 -30228.367} C_VEL
LIN {X 0,Y 144.641,Z 540.221,A -85,B 0,C 180,E1 -30228.649,E2 -30228.649} C_VEL
LIN {X 0,Y 145.935,Z 529.294,A -85,B 0,C 180,E1 -30228.892,E2 -30228.892} C_VEL
LIN {X 0,Y 145.568,Z 526.684,A -85,B 0,C 180,E1 -30233.066,E2 -30233.066} C_VEL
LIN {X 0,Y 145.618,Z 526.626,A -85,B 0,C 180,E1 -30237.059,E2 -30237.059} C_VEL
LIN {X 0,Y 145.903,Z 528.82,A -85,B 0,C 180,E1 -30240.344,E2 -30240.344} C_VEL
LIN {X 0,Y 145.973,Z 529.255,A -85,B 0,C 180,E1 -30240.832,E2 -30240.832} C_VEL
LIN {X 0,Y 143.053,Z 551.224,A -85,B 0,C 180,E1 -30241.199,E2 -30241.199} C_VEL
LIN {X 0,Y 139.643,Z 566.618,A -85,B 0,C 180,E1 -30241.547,E2 -30241.547} C_VEL
LIN {X 0,Y 134.926,Z 581.478,A -85,B 0,C 180,E1 -30241.921,E2 -30241.921} C_VEL
LIN {X 0,Y 129.252,Z 595.195,A -85,B 0,C 180,E1 -30242.385,E2 -30242.385} C_VEL
LIN {X 0,Y 123.156,Z 607.111,A -85,B 0,C 180,E1 -30243.001,E2 -30243.001} C_VEL
LIN {X 0,Y 115.362,Z 619.843,A -85,B 0,C 180,E1 -30243.974,E2 -30243.974} C_VEL
LIN {X 0,Y 109.305,Z 628.348,A -85,B 0,C 180,E1 -30244.714,E2 -30244.714} C_VEL
LIN {X 0,Y 98.995,Z 640.748,A -85,B 0,C 180,E1 -30246.321,E2 -30246.321} C_VEL
LIN {X 0,Y 88.774,Z 651.124,A -85,B 0,C 180,E1 -30248.272,E2 -30248.272} C_VEL
LIN {X 0,Y 77.041,Z 661.258,A -85,B 0,C 180,E1 -30251.285,E2 -30251.285} C_VEL
LIN {X 0,Y 65.599,Z 669.663,A -85,B 0,C 180,E1 -30255.369,E2 -30255.369} C_VEL
LIN {X 0,Y 53.063,Z 677.525,A -85,B 0,C 180,E1 -30262.007,E2 -30262.007} C_VEL
LIN {X 0,Y 41.637,Z 683.756,A -85,B 0,C 180,E1 -30272.437,E2 -30272.437} C_VEL
LIN {X 0,Y 32.37,Z 688.538,A -85,B 0,C 180,E1 -30289.356,E2 -30289.356} C_VEL
LIN {X 0,Y 27.381,Z 691.997,A -85,B 0,C 180,E1 -30315.126,E2 -30315.126} C_VEL
LIN {X 0,Y 27.106,Z 693.25,A -85,B 0,C 180,E1 -30329.999,E2 -30329.999} C_VEL
LIN {X 0,Y 27.459,Z 694.16,A -85,B 0,C 180,E1 -30344.829,E2 -30344.829} C_VEL
LIN {X 0,Y 32.468,Z 695.12,A -85,B 0,C 180,E1 -30370.494,E2 -30370.494} C_VEL
LIN {X 0,Y 41.836,Z 694.98,A -85,B 0,C 180,E1 -30387.135,E2 -30387.135} C_VEL
LIN {X 0,Y 53.356,Z 693.675,A -85,B 0,C 180,E1 -30397.224,E2 -30397.224} C_VEL
LIN {X 0,Y 65.955,Z 691.262,A -85,B 0,C 180,E1 -30403.538,E2 -30403.538} C_VEL
LIN {X 0,Y 79.092,Z 687.691,A -85,B 0,C 180,E1 -30407.808,E2 -30407.808} C_VEL
LIN {X 0,Y 92.529,Z 682.874,A -85,B 0,C 180,E1 -30410.899,E2 -30410.899} C_VEL
LIN {X 0,Y 106.188,Z 676.683,A -85,B 0,C 180,E1 -30413.105,E2 -30413.105} C_VEL
LIN {X 0,Y 119.983,Z 668.945,A -85,B 0,C 180,E1 -30414.731,E2 -30414.731} C_VEL
LIN {X 0,Y 126.908,Z 664.422,A -85,B 0,C 180,E1 -30415.424,E2 -30415.424} C_VEL
LIN {X 0,Y 126.789,Z 664.47,A -85,B 0,C 180,E1 -30416.16,E2 -30416.16} C_VEL
LIN {X 0,Y 119.355,Z 669.227,A -85,B 0,C 180,E1 -30417.016,E2 -30417.016} C_VEL
LIN {X 0,Y 113.198,Z 672.782,A -85,B 0,C 180,E1 -30417.435,E2 -30417.435} C_VEL
LIN {X 0,Y 102.563,Z 678.163,A -85,B 0,C 180,E1 -30417.319,E2 -30417.319} C_VEL
LIN {X 0,Y 93.847,Z 681.947,A -85,B 0,C 180,E1 -30417.17,E2 -30417.17} C_VEL
LIN {X 0,Y 87.246,Z 684.439,A -85,B 0,C 180,E1 -30417.556,E2 -30417.556} C_VEL
LIN {X 0,Y 85.067,Z 685.198,A -85,B 0,C 180,E1 -30417.87,E2 -30417.87} C_VEL
LIN {X 0,Y 70.292,Z 689.454,A -85,B 0,C 180,E1 -30421.069,E2 -30421.069} C_VEL
LIN {X 0,Y 56.494,Z 692.18,A -85,B 0,C 180,E1 -30425.606,E2 -30425.606} C_VEL
LIN {X 0,Y 43.25,Z 693.685,A -85,B 0,C 180,E1 -30432.843,E2 -30432.843} C_VEL
LIN {X 0,Y 29.895,Z 693.956,A -85,B 0,C 180,E1 -30448.052,E2 -30448.052} C_VEL
LIN {X 0,Y 22.099,Z 693.168,A -85,B 0,C 180,E1 -30470.504,E2 -30470.504} C_VEL
LIN {X 0,Y 19.872,Z 691.155,A -85,B 0,C 180,E1 -30510.001,E2 -30510.001} C_VEL
LIN {X 0,Y 22.473,Z 689.531,A -85,B 0,C 180,E1 -30530.228,E2 -30530.228} C_VEL
LIN {X 0,Y 30.431,Z 685.888,A -85,B 0,C 180,E1 -30553.857,E2 -30553.857} C_VEL
LIN {X 0,Y 41.659,Z 680.817,A -85,B 0,C 180,E1 -30567.515,E2 -30567.515} C_VEL
LIN {X 0,Y 54.187,Z 674.322,A -85,B 0,C 180,E1 -30575.216,E2 -30575.216} C_VEL
LIN {X 0,Y 67.25,Z 666.218,A -85,B 0,C 180,E1 -30580.145,E2 -30580.145} C_VEL
LIN {X 0,Y 78.931,Z 657.575,A -85,B 0,C 180,E1 -30583.175,E2 -30583.175} C_VEL
LIN {X 0,Y 90.762,Z 647.186,A -85,B 0,C 180,E1 -30585.448,E2 -30585.448} C_VEL
LIN {X 0,Y 100.989,Z 636.525,A -85,B 0,C 180,E1 -30586.98,E2 -30586.98} C_VEL
LIN {X 0,Y 111.263,Z 623.741,A -85,B 0,C 180,E1 -30588.258,E2 -30588.258} C_VEL
LIN {X 0,Y 119.85,Z 610.834,A -85,B 0,C 180,E1 -30589.182,E2 -30589.182} C_VEL
LIN {X 0,Y 127.589,Z 596.577,A -85,B 0,C 180,E1 -30589.937,E2 -30589.937} C_VEL
LIN {X 0,Y 133.601,Z 582.646,A -85,B 0,C 180,E1 -30590.518,E2 -30590.518} C_VEL
LIN {X 0,Y 138.664,Z 567.337,A -85,B 0,C 180,E1 -30590.957,E2 -30590.957} C_VEL
LIN {X 0,Y 142.208,Z 552.174,A -85,B 0,C 180,E1 -30591.272,E2 -30591.272} C_VEL
LIN {X 0,Y 144.719,Z 534.823,A -85,B 0,C 180,E1 -30591.565,E2 -30591.565} C_VEL
LIN {X 0,Y 144.674,Z 533.61,A -85,B 0,C 180,E1 -30593.724,E2 -30593.724} C_VEL
LIN {X 0,Y 144.717,Z 533.654,A -85,B 0,C 180,E1 -30596.693,E2 -30596.693} C_VEL
LIN {X 0,Y 144.77,Z 534.513,A -85,B 0,C 180,E1 -30598.125,E2 -30598.125} C_VEL
LIN {X 0,Y 142.125,Z 552.832,A -85,B 0,C 180,E1 -30598.382,E2 -30598.382} C_VEL
LIN {X 0,Y 138.441,Z 568.446,A -85,B 0,C 180,E1 -30598.677,E2 -30598.677} C_VEL
LIN {X 0,Y 133.554,Z 583.125,A -85,B 0,C 180,E1 -30598.975,E2 -30598.975} C_VEL
LIN {X 0,Y 127.392,Z 597.329,A -85,B 0,C 180,E1 -30599.336,E2 -30599.336} C_VEL
LIN {X 0,Y 122.114,Z 607.386,A -85,B 0,C 180,E1 -30599.727,E2 -30599.727} C_VEL
LIN {X 0,Y 114.006,Z 620.337,A -85,B 0,C 180,E1 -30600.504,E2 -30600.504} C_VEL
LIN {X 0,Y 107.199,Z 629.569,A -85,B 0,C 180,E1 -30601.15,E2 -30601.15} C_VEL
LIN {X 0,Y 98.461,Z 639.88,A -85,B 0,C 180,E1 -30602.136,E2 -30602.136} C_VEL
LIN {X 0,Y 88.029,Z 650.339,A -85,B 0,C 180,E1 -30603.648,E2 -30603.648} C_VEL
LIN {X 0,Y 77.664,Z 659.18,A -85,B 0,C 180,E1 -30605.486,E2 -30605.486} C_VEL
LIN {X 0,Y 65.761,Z 667.918,A -85,B 0,C 180,E1 -30608.669,E2 -30608.669} C_VEL
LIN {X 0,Y 54.079,Z 675.148,A -85,B 0,C 180,E1 -30612.915,E2 -30612.915} C_VEL
LIN {X 0,Y 41.043,Z 681.955,A -85,B 0,C 180,E1 -30620.812,E2 -30620.812} C_VEL
LIN {X 0,Y 29.831,Z 687.048,A -85,B 0,C 180,E1 -30634.453,E2 -30634.453} C_VEL
LIN {X 0,Y 23.164,Z 690.052,A -85,B 0,C 180,E1 -30652.64,E2 -30652.64} C_VEL
LIN {X 0,Y 19.991,Z 692.934,A -85,B 0,C 180,E1 -30689.999,E2 -30689.999} C_VEL
LIN {X 0,Y 20.636,Z 693.871,A -85,B 0,C 180,E1 -30709.91,E2 -30709.91} C_VEL
LIN {X 0,Y 27.421,Z 694.886,A -85,B 0,C 180,E1 -30740.253,E2 -30740.253} C_VEL
LIN {X 0,Y 38.419,Z 694.776,A -85,B 0,C 180,E1 -30756.156,E2 -30756.156} C_VEL
LIN {X 0,Y 51.016,Z 693.524,A -85,B 0,C 180,E1 -30764.65,E2 -30764.65} C_VEL
LIN {X 0,Y 64.291,Z 691.167,A -85,B 0,C 180,E1 -30769.686,E2 -30769.686} C_VEL
LIN {X 0,Y 77.895,Z 687.654,A -85,B 0,C 180,E1 -30772.963,E2 -30772.963} C_VEL
LIN {X 0,Y 91.669,Z 682.899,A -85,B 0,C 180,E1 -30775.323,E2 -30775.323} C_VEL
LIN {X 0,Y 94.455,Z 681.748,A -85,B 0,C 180,E1 -30775.735,E2 -30775.735} C_VEL
LIN {X 0,Y 91.504,Z 682.909,A -85,B 0,C 180,E1 -30776.825,E2 -30776.825} C_VEL
LIN {X 0,Y 85.067,Z 685.198,A -85,B 0,C 180,E1 -30777.87,E2 -30777.87} C_VEL
LIN {X 0,Y 79.271,Z 687.09,A -85,B 0,C 180,E1 -30778.46,E2 -30778.46} C_VEL
LIN {X 0,Y 69.301,Z 689.752,A -85,B 0,C 180,E1 -30778.253,E2 -30778.253} C_VEL
LIN {X 0,Y 61.214,Z 691.478,A -85,B 0,C 180,E1 -30777.95,E2 -30777.95} C_VEL
LIN {X 0,Y 55.162,Z 692.472,A -85,B 0,C 180,E1 -30778.481,E2 -30778.481} C_VEL
LIN {X 0,Y 53.181,Z 692.715,A -85,B 0,C 180,E1 -30778.962,E2 -30778.962} C_VEL
LIN {X 0,Y 42.228,Z 693.868,A -85,B 0,C 180,E1 -30783.051,E2 -30783.051} C_VEL
LIN {X 0,Y 28.797,Z 694.247,A -85,B 0,C 180,E1 -30792.522,E2 -30792.522} C_VEL
LIN {X 0,Y 17.126,Z 693.463,A -85,B 0,C 180,E1 -30814.844,E2 -30814.844} C_VEL
LIN {X 0,Y 12.671,Z 691.478,A -85,B 0,C 180,E1 -30870.002,E2 -30870.002} C_VEL
LIN {X 0,Y 16.604,Z 689.65,A -85,B 0,C 180,E1 -30902.142,E2 -30902.142} C_VEL
LIN {X 0,Y 28.812,Z 685.195,A -85,B 0,C 180,E1 -30928.621,E2 -30928.621} C_VEL
LIN {X 0,Y 41.605,Z 679.862,A -85,B 0,C 180,E1 -30938.293,E2 -30938.293} C_VEL
LIN {X 0,Y 55.007,Z 673.054,A -85,B 0,C 180,E1 -30943.386,E2 -30943.386} C_VEL
LIN {X 0,Y 68.608,Z 664.584,A -85,B 0,C 180,E1 -30946.696,E2 -30946.696} C_VEL
LIN {X 0,Y 80.623,Z 655.574,A -85,B 0,C 180,E1 -30948.72,E2 -30948.72} C_VEL
LIN {X 0,Y 92.716,Z 644.703,A -85,B 0,C 180,E1 -30950.206,E2 -30950.206} C_VEL
LIN {X 0,Y 103.105,Z 633.538,A -85,B 0,C 180,E1 -30951.258,E2 -30951.258} C_VEL
LIN {X 0,Y 112.654,Z 621.277,A -85,B 0,C 180,E1 -30952.048,E2 -30952.048} C_VEL
LIN {X 0,Y 121.335,Z 607.788,A -85,B 0,C 180,E1 -30952.715,E2 -30952.715} C_VEL
LIN {X 0,Y 128.286,Z 594.542,A -85,B 0,C 180,E1 -30953.199,E2 -30953.199} C_VEL
LIN {X 0,Y 134.359,Z 579.99,A -85,B 0,C 180,E1 -30953.641,E2 -30953.641} C_VEL
LIN {X 0,Y 139.27,Z 564.341,A -85,B 0,C 180,E1 -30953.959,E2 -30953.959} C_VEL
LIN {X 0,Y 142.675,Z 548.378,A -85,B 0,C 180,E1 -30954.193,E2 -30954.193} C_VEL
LIN {X 0,Y 143.794,Z 540.583,A -85,B 0,C 180,E1 -30954.332,E2 -30954.332} C_VEL
LIN {X 0,Y 143.801,Z 540.523,A -85,B 0,C 180,E1 -30955.374,E2 -30955.374} C_VEL
LIN {X 0,Y 141.202,Z 556.221,A -85,B 0,C 180,E1 -30955.574,E2 -30955.574} C_VEL
LIN {X 0,Y 137.471,Z 570.692,A -85,B 0,C 180,E1 -30955.753,E2 -30955.753} C_VEL
LIN {X 0,Y 132.548,Z 584.751,A -85,B 0,C 180,E1 -30955.937,E2 -30955.937} C_VEL
LIN {X 0,Y 126.79,Z 597.67,A -85,B 0,C 180,E1 -30956.157,E2 -30956.157} C_VEL
LIN {X 0,Y 121.473,Z 607.667,A -85,B 0,C 180,E1 -30956.407,E2 -30956.407} C_VEL
LIN {X 0,Y 112.606,Z 621.518,A -85,B 0,C 180,E1 -30956.975,E2 -30956.975} C_VEL
LIN {X 0,Y 102.873,Z 634.023,A -85,B 0,C 180,E1 -30957.634,E2 -30957.634} C_VEL
LIN {X 0,Y 91.392,Z 646.241,A -85,B 0,C 180,E1 -30958.595,E2 -30958.595} C_VEL
LIN {X 0,Y 80.472,Z 656.004,A -85,B 0,C 180,E1 -30959.797,E2 -30959.797} C_VEL
LIN {X 0,Y 68.554,Z 664.99,A -85,B 0,C 180,E1 -30961.709,E2 -30961.709} C_VEL
LIN {X 0,Y 56.385,Z 672.668,A -85,B 0,C 180,E1 -30964.318,E2 -30964.318} C_VEL
LIN {X 0,Y 42.703,Z 679.828,A -85,B 0,C 180,E1 -30969.072,E2 -30969.072} C_VEL
LIN {X 0,Y 29.565,Z 685.448,A -85,B 0,C 180,E1 -30978.034,E2 -30978.034} C_VEL
LIN {X 0,Y 18.008,Z 689.677,A -85,B 0,C 180,E1 -30998.688,E2 -30998.688} C_VEL
LIN {X 0,Y 12.89,Z 692.619,A -85,B 0,C 180,E1 -31049.998,E2 -31049.998} C_VEL
LIN {X 0,Y 14.143,Z 693.582,A -85,B 0,C 180,E1 -31079.796,E2 -31079.796} C_VEL
LIN {X 0,Y 23.497,Z 694.651,A -85,B 0,C 180,E1 -31113.802,E2 -31113.802} C_VEL
LIN {X 0,Y 36.122,Z 694.569,A -85,B 0,C 180,E1 -31126.611,E2 -31126.611} C_VEL
LIN {X 0,Y 49.602,Z 693.372,A -85,B 0,C 180,E1 -31132.658,E2 -31132.658} C_VEL
LIN {X 0,Y 63.4,Z 691.071,A -85,B 0,C 180,E1 -31136.077,E2 -31136.077} C_VEL
LIN {X 0,Y 63.376,Z 691.066,A -85,B 0,C 180,E1 -31136.405,E2 -31136.405} C_VEL
LIN {X 0,Y 53.181,Z 692.715,A -85,B 0,C 180,E1 -31138.962,E2 -31138.962} C_VEL
LIN {X 0,Y 46.688,Z 693.528,A -85,B 0,C 180,E1 -31140.333,E2 -31140.333} C_VEL
LIN {X 0,Y 35.586,Z 694.301,A -85,B 0,C 180,E1 -31140.848,E2 -31140.848} C_VEL
LIN {X 0,Y 26.644,Z 694.414,A -85,B 0,C 180,E1 -31141.06,E2 -31141.06} C_VEL
LIN {X 0,Y 20.033,Z 694.185,A -85,B 0,C 180,E1 -31143.259,E2 -31143.259} C_VEL
LIN {X 0,Y 17.896,Z 694.026,A -85,B 0,C 180,E1 -31145.084,E2 -31145.084} C_VEL
LIN {X 0,Y 8.124,Z 692.919,A -85,B 0,C 180,E1 -31170.113,E2 -31170.113} C_VEL
LIN {X 0,Y 9.666,Z 690.392,A -85,B 0,C 180,E1 -31276.646,E2 -31276.646} C_VEL
LIN {X 0,Y 15.843,Z 688.7,A -85,B 0,C 180,E1 -31292.529,E2 -31292.529} C_VEL
LIN {X 0,Y 29.237,Z 684.398,A -85,B 0,C 180,E1 -31304.056,E2 -31304.056} C_VEL
LIN {X 0,Y 42.992,Z 678.769,A -85,B 0,C 180,E1 -31308.766,E2 -31308.766} C_VEL
LIN {X 0,Y 56.89,Z 671.637,A -85,B 0,C 180,E1 -31311.23,E2 -31311.23} C_VEL
LIN {X 0,Y 69.079,Z 664.013,A -85,B 0,C 180,E1 -31312.733,E2 -31312.733} C_VEL
LIN {X 0,Y 81.291,Z 654.851,A -85,B 0,C 180,E1 -31313.847,E2 -31313.847} C_VEL
LIN {X 0,Y 84.785,Z 651.895,A -85,B 0,C 180,E1 -31314.105,E2 -31314.105} C_VEL
LIN {X 0,Y 84.731,Z 651.951,A -85,B 0,C 180,E1 -31314.469,E2 -31314.469} C_VEL
LIN {X 0,Y 72.268,Z 661.831,A -85,B 0,C 180,E1 -31315.33,E2 -31315.33} C_VEL
